LIN {X 0.167,Y -651.336,Z 1359.331,A 0.000,B 0.000,C 90.000,E1 95.511} C_DIS
LIN {X 0.159,Y -645.821,Z 1359.326,A 0.000,B 0.000,C 90.000,E1 94.645} C_DIS
LIN {X 0.149,Y -640.696,Z 1359.322,A 0.000,B 0.000,C 90.000,E1 93.898} C_DIS
LIN {X 0.299,Y -636.929,Z 1359.319,A 0.000,B 0.000,C 90.000,E1 93.383} C_DIS
LIN {X -0.288,Y -631.276,Z 1359.316,A 0.000,B 0.000,C 90.000,E1 92.808} C_DIS
LIN {X -0.177,Y -625.115,Z 1359.312,A 0.000,B 0.000,C 90.000,E1 92.178} C_DIS
LIN {X -0.172,Y -616.219,Z 1359.307,A 0.000,B 0.000,C 90.000,E1 91.318} C_DIS
LIN {X 0.233,Y -610.785,Z 1359.305,A 0.000,B 0.000,C 90.000,E1 90.802} C_DIS
LIN {X 0.209,Y -607.830,Z 1359.303,A 0.000,B 0.000,C 90.000,E1 90.573} C_DIS
LIN {X -0.246,Y -603.158,Z 1359.302,A 0.000,B 0.000,C 90.000,E1 90.286} C_DIS
LIN {X -0.039,Y -596.420,Z 1359.299,A 0.000,B 0.000,C 90.000,E1 89.885} C_DIS
LIN {X -0.028,Y -592.860,Z 1359.298,A 0.000,B 0.000,C 90.000,E1 89.714} C_DIS
LIN {X -0.153,Y -585.830,Z 1359.297,A 0.000,B 0.000,C 90.000,E1 89.427} C_DIS
LIN {X 0.188,Y -582.520,Z 1359.296,A 0.000,B 0.000,C 90.000,E1 89.255} C_DIS
LIN {X -0.070,Y -578.389,Z 1359.295,A 0.000,B 0.000,C 90.000,E1 89.083} C_DIS
LIN {X 0.000,Y -574.152,Z 1359.293,A 0.000,B 0.000,C 90.000,E1 88.797} C_DIS
LIN {X -0.034,Y -574.128,Z 1359.293,A 0.000,B 0.000,C 90.000,E1 88.797} C_DIS
LIN {X 0.004,Y -573.399,Z 1359.292,A 0.000,B 0.000,C 90.000,E1 88.625} C_DIS
LIN {X -0.160,Y -573.188,Z 1359.290,A 0.000,B 0.000,C 90.000,E1 88.165} C_DIS
LIN {X 0.226,Y -575.527,Z 1359.275,A 0.000,B 0.000,C 90.000,E1 85.412} C_DIS
LIN {X 0.222,Y -577.636,Z 1359.264,A 0.000,B 0.000,C 90.000,E1 83.514} C_DIS
LIN {X -0.164,Y -579.848,Z 1359.254,A 0.000,B 0.000,C 90.000,E1 81.659} C_DIS
LIN {X 0.201,Y -581.498,Z 1359.246,A 0.000,B 0.000,C 90.000,E1 80.274} C_DIS
LIN {X 0.218,Y -582.949,Z 1359.239,A 0.000,B 0.000,C 90.000,E1 78.926} C_DIS
LIN {X -0.092,Y -584.010,Z 1359.233,A 0.000,B 0.000,C 90.000,E1 77.881} C_DIS
LIN {X -0.220,Y -585.490,Z 1359.224,A 0.000,B 0.000,C 90.000,E1 76.284} C_DIS
LIN {X -0.138,Y -586.504,Z 1359.216,A 0.000,B 0.000,C 90.000,E1 74.936} C_DIS
LIN {X -0.144,Y -587.223,Z 1359.210,A 0.000,B 0.000,C 90.000,E1 73.866} C_DIS
LIN {X -0.199,Y -588.435,Z 1359.200,A 0.000,B 0.000,C 90.000,E1 72.000} C_DIS
LIN {X 0.200,Y -589.644,Z 1359.188,A 0.000,B 0.000,C 90.000,E1 69.826} C_DIS
LIN {X -0.062,Y -590.952,Z 1359.176,A 0.000,B 0.000,C 90.000,E1 67.720} C_DIS
LIN {X 0.061,Y -592.317,Z 1359.166,A 0.000,B 0.000,C 90.000,E1 65.845} C_DIS
LIN {X -0.139,Y -593.439,Z 1359.159,A 0.000,B 0.000,C 90.000,E1 64.537} C_DIS
LIN {X 0.099,Y -594.582,Z 1359.150,A 0.000,B 0.000,C 90.000,E1 62.922} C_DIS
LIN {X 0.280,Y -596.052,Z 1359.139,A 0.000,B 0.000,C 90.000,E1 61.051} C_DIS
LIN {X 0.132,Y -597.309,Z 1359.132,A 0.000,B 0.000,C 90.000,E1 59.744} C_DIS
LIN {X -0.208,Y -598.613,Z 1359.125,A 0.000,B 0.000,C 90.000,E1 58.456} C_DIS
LIN {X 0.220,Y -600.158,Z 1359.116,A 0.000,B 0.000,C 90.000,E1 56.834} C_DIS
LIN {X 0.018,Y -601.130,Z 1359.110,A 0.000,B 0.000,C 90.000,E1 55.801} C_DIS
LIN {X 0.327,Y -602.568,Z 1359.101,A 0.000,B 0.000,C 90.000,E1 54.196} C_DIS
LIN {X -0.341,Y -603.576,Z 1359.095,A 0.000,B 0.000,C 90.000,E1 53.210} C_DIS
LIN {X 0.213,Y -604.481,Z 1359.090,A 0.000,B 0.000,C 90.000,E1 52.110} C_DIS
LIN {X 0.196,Y -605.361,Z 1359.082,A 0.000,B 0.000,C 90.000,E1 50.803} C_DIS
LIN {X -0.282,Y -606.128,Z 1359.075,A 0.000,B 0.000,C 90.000,E1 49.542} C_DIS
LIN {X -0.159,Y -606.615,Z 1359.069,A 0.000,B 0.000,C 90.000,E1 48.485} C_DIS
LIN {X -0.007,Y -607.015,Z 1359.061,A 0.000,B 0.000,C 90.000,E1 46.905} C_DIS
LIN {X 0.160,Y -607.095,Z 1359.052,A 0.000,B 0.000,C 90.000,E1 45.324} C_DIS
LIN {X 0.266,Y -607.003,Z 1359.046,A 0.000,B 0.000,C 90.000,E1 44.271} C_DIS
LIN {X -0.051,Y -606.655,Z 1359.040,A 0.000,B 0.000,C 90.000,E1 43.257} C_DIS
LIN {X 0.100,Y -605.947,Z 1359.032,A 0.000,B 0.000,C 90.000,E1 41.676} C_DIS
LIN {X 0.220,Y -605.426,Z 1359.026,A 0.000,B 0.000,C 90.000,E1 40.620} C_DIS
LIN {X 0.004,Y -604.489,Z 1359.017,A 0.000,B 0.000,C 90.000,E1 39.072} C_DIS
LIN {X 0.356,Y -603.496,Z 1359.010,A 0.000,B 0.000,C 90.000,E1 37.729} C_DIS
LIN {X 0.283,Y -602.735,Z 1359.005,A 0.000,B 0.000,C 90.000,E1 36.950} C_DIS
LIN {X 0.206,Y -601.887,Z 1359.001,A 0.000,B 0.000,C 90.000,E1 36.171} C_DIS
LIN {X 0.120,Y -600.627,Z 1358.997,A 0.000,B 0.000,C 90.000,E1 35.391} C_DIS
LIN {X 0.019,Y -599.217,Z 1358.992,A 0.000,B 0.000,C 90.000,E1 34.612} C_DIS
LIN {X -0.200,Y -597.011,Z 1358.986,A 0.000,B 0.000,C 90.000,E1 33.579} C_DIS
LIN {X 0.269,Y -593.830,Z 1358.979,A 0.000,B 0.000,C 90.000,E1 32.212} C_DIS
LIN {X -0.129,Y -592.363,Z 1358.976,A 0.000,B 0.000,C 90.000,E1 31.720} C_DIS
LIN {X -0.253,Y -588.851,Z 1358.970,A 0.000,B 0.000,C 90.000,E1 30.669} C_DIS
LIN {X -0.299,Y -585.983,Z 1358.966,A 0.000,B 0.000,C 90.000,E1 29.873} C_DIS
LIN {X -0.250,Y -583.870,Z 1358.963,A 0.000,B 0.000,C 90.000,E1 29.333} C_DIS
LIN {X 0.157,Y -580.292,Z 1358.958,A 0.000,B 0.000,C 90.000,E1 28.487} C_DIS
LIN {X -0.066,Y -575.633,Z 1358.953,A 0.000,B 0.000,C 90.000,E1 27.564} C_DIS
LIN {X 0.060,Y -572.066,Z 1358.949,A 0.000,B 0.000,C 90.000,E1 26.873} C_DIS
LIN {X -0.266,Y -568.990,Z 1358.946,A 0.000,B 0.000,C 90.000,E1 26.360} C_DIS
LIN {X -0.191,Y -564.804,Z 1358.943,A 0.000,B 0.000,C 90.000,E1 25.668} C_DIS
LIN {X 0.184,Y -561.209,Z 1358.939,A 0.000,B 0.000,C 90.000,E1 25.079} C_DIS
LIN {X -0.103,Y -558.437,Z 1358.937,A 0.000,B 0.000,C 90.000,E1 24.695} C_DIS
LIN {X -0.125,Y -553.412,Z 1358.933,A 0.000,B 0.000,C 90.000,E1 24.003} C_DIS
LIN {X -0.023,Y -546.987,Z 1358.929,A 0.000,B 0.000,C 90.000,E1 23.153} C_DIS
LIN {X -0.015,Y -542.308,Z 1358.926,A 0.000,B 0.000,C 90.000,E1 22.589} C_DIS
LIN {X 0.297,Y -534.020,Z 1358.920,A 0.000,B 0.000,C 90.000,E1 21.589} C_DIS
LIN {X 0.096,Y -523.631,Z 1358.914,A 0.000,B 0.000,C 90.000,E1 20.482} C_DIS
LIN {X -0.092,Y -513.039,Z 1358.908,A 0.000,B 0.000,C 90.000,E1 19.396} C_DIS
LIN {X 0.217,Y -502.297,Z 1358.901,A 0.000,B 0.000,C 90.000,E1 18.236} C_DIS
LIN {X 0.199,Y -493.019,Z 1358.896,A 0.000,B 0.000,C 90.000,E1 17.275} C_DIS
LIN {X 0.067,Y -480.292,Z 1358.889,A 0.000,B 0.000,C 90.000,E1 16.079} C_DIS
LIN {X 0.101,Y -467.549,Z 1358.882,A 0.000,B 0.000,C 90.000,E1 14.828} C_DIS
LIN {X 0.172,Y -457.530,Z 1358.877,A 0.000,B 0.000,C 90.000,E1 13.828} C_DIS
LIN {X 0.113,Y -438.983,Z 1358.867,A 0.000,B 0.000,C 90.000,E1 11.951} C_DIS
LIN {X 0.208,Y -420.924,Z 1358.856,A 0.000,B 0.000,C 90.000,E1 9.962} C_DIS
LIN {X -0.132,Y -406.834,Z 1358.847,A 0.000,B 0.000,C 90.000,E1 8.398} C_DIS
LIN {X 0.062,Y -397.118,Z 1358.840,A 0.000,B 0.000,C 90.000,E1 7.239} C_DIS
LIN {X -0.114,Y -393.534,Z 1358.837,A 0.000,B 0.000,C 90.000,E1 6.720} C_DIS
LIN {X -0.153,Y -393.499,Z 1358.837,A 0.000,B 0.000,C 90.000,E1 6.720} C_DIS
LIN {X 0.105,Y -395.070,Z 1358.836,A 0.000,B 0.000,C 90.000,E1 6.429} C_DIS
LIN {X -0.156,Y -397.982,Z 1358.834,A 0.000,B 0.000,C 90.000,E1 6.201} C_DIS
LIN {X -0.095,Y -401.724,Z 1358.833,A 0.000,B 0.000,C 90.000,E1 5.910} C_DIS
LIN {X -0.107,Y -410.009,Z 1358.830,A 0.000,B 0.000,C 90.000,E1 5.334} C_DIS
LIN {X 0.013,Y -417.658,Z 1358.826,A 0.000,B 0.000,C 90.000,E1 4.702} C_DIS
LIN {X -0.174,Y -423.633,Z 1358.823,A 0.000,B 0.000,C 90.000,E1 4.188} C_DIS
LIN {X -0.069,Y -430.586,Z 1358.819,A 0.000,B 0.000,C 90.000,E1 3.440} C_DIS
LIN {X 0.124,Y -437.371,Z 1358.815,A 0.000,B 0.000,C 90.000,E1 2.636} C_DIS
LIN {X -0.030,Y -442.782,Z 1358.811,A 0.000,B 0.000,C 90.000,E1 2.007} C_DIS
LIN {X -0.066,Y -450.455,Z 1358.806,A 0.000,B 0.000,C 90.000,E1 1.031} C_DIS
LIN {X 0.000,Y -457.754,Z 1358.800,A 0.000,B 0.000,C 90.000,E1 360.000} C_DIS
LIN {X 0.008,Y -462.424,Z 1358.796,A 0.000,B 0.000,C 90.000,E1 359.312} C_DIS
LIN {X 0.077,Y -467.489,Z 1358.792,A 0.000,B 0.000,C 90.000,E1 358.511} C_DIS
LIN {X 0.212,Y -472.140,Z 1358.787,A 0.000,B 0.000,C 90.000,E1 357.707} C_DIS
LIN {X -0.104,Y -476.442,Z 1358.783,A 0.000,B 0.000,C 90.000,E1 356.963} C_DIS
LIN {X -0.018,Y -479.732,Z 1358.780,A 0.000,B 0.000,C 90.000,E1 356.331} C_DIS
LIN {X -0.095,Y -484.122,Z 1358.775,A 0.000,B 0.000,C 90.000,E1 355.412} C_DIS
LIN {X 0.206,Y -487.474,Z 1358.770,A 0.000,B 0.000,C 90.000,E1 354.609} C_DIS
LIN {X 0.226,Y -489.412,Z 1358.768,A 0.000,B 0.000,C 90.000,E1 354.147} C_DIS
LIN {X -0.190,Y -492.808,Z 1358.763,A 0.000,B 0.000,C 90.000,E1 353.280} C_DIS
LIN {X 0.022,Y -494.928,Z 1358.759,A 0.000,B 0.000,C 90.000,E1 352.648} C_DIS
LIN {X -0.176,Y -496.874,Z 1358.756,A 0.000,B 0.000,C 90.000,E1 352.064} C_DIS
LIN {X -0.020,Y -499.436,Z 1358.751,A 0.000,B 0.000,C 90.000,E1 351.141} C_DIS
LIN {X 0.088,Y -502.578,Z 1358.744,A 0.000,B 0.000,C 90.000,E1 349.926} C_DIS
LIN {X -0.109,Y -504.658,Z 1358.739,A 0.000,B 0.000,C 90.000,E1 349.050} C_DIS
LIN {X -0.282,Y -506.462,Z 1358.734,A 0.000,B 0.000,C 90.000,E1 348.173} C_DIS
LIN {X 0.168,Y -508.137,Z 1358.729,A 0.000,B 0.000,C 90.000,E1 347.229} C_DIS
LIN {X 0.069,Y -510.411,Z 1358.721,A 0.000,B 0.000,C 90.000,E1 345.755} C_DIS
LIN {X 0.079,Y -511.492,Z 1358.716,A 0.000,B 0.000,C 90.000,E1 344.866} C_DIS
LIN {X 0.100,Y -512.345,Z 1358.711,A 0.000,B 0.000,C 90.000,E1 343.976} C_DIS
LIN {X 0.126,Y -512.947,Z 1358.706,A 0.000,B 0.000,C 90.000,E1 343.087} C_DIS
LIN {X 0.236,Y -513.014,Z 1358.704,A 0.000,B 0.000,C 90.000,E1 342.779} C_DIS
LIN {X 0.194,Y -512.921,Z 1358.703,A 0.000,B 0.000,C 90.000,E1 342.489} C_DIS
LIN {X -0.182,Y -512.687,Z 1358.701,A 0.000,B 0.000,C 90.000,E1 342.236} C_DIS
LIN {X -0.226,Y -512.193,Z 1358.700,A 0.000,B 0.000,C 90.000,E1 341.945} C_DIS
LIN {X -0.112,Y -511.312,Z 1358.698,A 0.000,B 0.000,C 90.000,E1 341.638} C_DIS
LIN {X 0.186,Y -510.592,Z 1358.697,A 0.000,B 0.000,C 90.000,E1 341.456} C_DIS
LIN {X 0.001,Y -509.317,Z 1358.696,A 0.000,B 0.000,C 90.000,E1 341.329} C_DIS
LIN {X -0.056,Y -501.855,Z 1358.695,A 0.000,B 0.000,C 90.000,E1 341.040} C_DIS
LIN {X 0.071,Y -471.003,Z 1358.688,A 0.000,B 0.000,C 90.000,E1 339.752} C_DIS
LIN {X -0.074,Y -442.137,Z 1358.680,A 0.000,B 0.000,C 90.000,E1 338.411} C_DIS
LIN {X -0.024,Y -416.847,Z 1358.672,A 0.000,B 0.000,C 90.000,E1 337.050} C_DIS
LIN {X 0.105,Y -393.487,Z 1358.665,A 0.000,B 0.000,C 90.000,E1 335.613} C_DIS
LIN {X 0.028,Y -372.048,Z 1358.656,A 0.000,B 0.000,C 90.000,E1 334.152} C_DIS
LIN {X -0.045,Y -364.343,Z 1358.653,A 0.000,B 0.000,C 90.000,E1 333.589} C_DIS
LIN {X -0.070,Y -364.332,Z 1358.653,A 0.000,B 0.000,C 90.000,E1 333.589} C_DIS
LIN {X -0.037,Y -365.965,Z 1358.643,A 0.000,B 0.000,C 90.000,E1 331.691} C_DIS
LIN {X 0.125,Y -366.381,Z 1358.639,A 0.000,B 0.000,C 90.000,E1 330.923} C_DIS
LIN {X 0.067,Y -371.337,Z 1358.604,A 0.000,B 0.000,C 90.000,E1 324.642} C_DIS
LIN {X 0.055,Y -371.755,Z 1358.602,A 0.000,B 0.000,C 90.000,E1 324.276} C_DIS
LIN {X -0.169,Y -377.338,Z 1358.567,A 0.000,B 0.000,C 90.000,E1 318.081} C_DIS
LIN {X 0.111,Y -378.225,Z 1358.563,A 0.000,B 0.000,C 90.000,E1 317.310} C_DIS
LIN {X 0.101,Y -383.920,Z 1358.531,A 0.000,B 0.000,C 90.000,E1 311.515} C_DIS
LIN {X -0.104,Y -384.881,Z 1358.527,A 0.000,B 0.000,C 90.000,E1 310.825} C_DIS
LIN {X -0.183,Y -390.590,Z 1358.495,A 0.000,B 0.000,C 90.000,E1 305.105} C_DIS
LIN {X -0.117,Y -391.084,Z 1358.493,A 0.000,B 0.000,C 90.000,E1 304.739} C_DIS
LIN {X 0.123,Y -391.639,Z 1358.489,A 0.000,B 0.000,C 90.000,E1 303.992} C_DIS
LIN {X 0.019,Y -396.807,Z 1358.459,A 0.000,B 0.000,C 90.000,E1 298.693} C_DIS
LIN {X -0.110,Y -397.114,Z 1358.458,A 0.000,B 0.000,C 90.000,E1 298.359} C_DIS
LIN {X 0.045,Y -401.585,Z 1358.426,A 0.000,B 0.000,C 90.000,E1 292.717} C_DIS
LIN {X -0.064,Y -404.646,Z 1358.395,A 0.000,B 0.000,C 90.000,E1 287.149} C_DIS
LIN {X 0.022,Y -404.736,Z 1358.391,A 0.000,B 0.000,C 90.000,E1 286.441} C_DIS
LIN {X -0.082,Y -406.092,Z 1358.364,A 0.000,B 0.000,C 90.000,E1 281.591} C_DIS
LIN {X -0.075,Y -406.100,Z 1358.362,A 0.000,B 0.000,C 90.000,E1 281.243} C_DIS
LIN {X -0.039,Y -405.676,Z 1358.333,A 0.000,B 0.000,C 90.000,E1 276.030} C_DIS
LIN {X -0.030,Y -405.294,Z 1358.330,A 0.000,B 0.000,C 90.000,E1 275.334} C_DIS
LIN {X 0.040,Y -403.505,Z 1358.305,A 0.000,B 0.000,C 90.000,E1 270.802} C_DIS
LIN {X 0.008,Y -403.297,Z 1358.303,A 0.000,B 0.000,C 90.000,E1 270.458} C_DIS
LIN {X 0.191,Y -398.946,Z 1358.271,A 0.000,B 0.000,C 90.000,E1 264.837} C_DIS
LIN {X 0.059,Y -393.120,Z 1358.242,A 0.000,B 0.000,C 90.000,E1 259.567} C_DIS
LIN {X 0.020,Y -392.850,Z 1358.240,A 0.000,B 0.000,C 90.000,E1 259.218} C_DIS
LIN {X 0.133,Y -386.009,Z 1358.212,A 0.000,B 0.000,C 90.000,E1 254.212} C_DIS
LIN {X 0.074,Y -385.282,Z 1358.208,A 0.000,B 0.000,C 90.000,E1 253.504} C_DIS
LIN {X 0.094,Y -384.794,Z 1358.206,A 0.000,B 0.000,C 90.000,E1 253.142} C_DIS
LIN {X -0.033,Y -377.991,Z 1358.182,A 0.000,B 0.000,C 90.000,E1 248.827} C_DIS
LIN {X 0.054,Y -376.249,Z 1358.174,A 0.000,B 0.000,C 90.000,E1 247.358} C_DIS
LIN {X 0.155,Y -374.973,Z 1358.170,A 0.000,B 0.000,C 90.000,E1 246.613} C_DIS
LIN {X -0.110,Y -368.437,Z 1358.148,A 0.000,B 0.000,C 90.000,E1 242.615} C_DIS
LIN {X 0.193,Y -366.076,Z 1358.138,A 0.000,B 0.000,C 90.000,E1 240.717} C_DIS
LIN {X 0.100,Y -359.217,Z 1358.115,A 0.000,B 0.000,C 90.000,E1 236.628} C_DIS
LIN {X 0.117,Y -355.870,Z 1358.100,A 0.000,B 0.000,C 90.000,E1 233.989} C_DIS
LIN {X -0.078,Y -348.813,Z 1358.075,A 0.000,B 0.000,C 90.000,E1 229.461} C_DIS
LIN {X -0.002,Y -346.201,Z 1358.062,A 0.000,B 0.000,C 90.000,E1 227.148} C_DIS
LIN {X -0.115,Y -345.709,Z 1358.060,A 0.000,B 0.000,C 90.000,E1 226.782} C_DIS
LIN {X -0.153,Y -339.000,Z 1358.032,A 0.000,B 0.000,C 90.000,E1 221.757} C_DIS
LIN {X -0.073,Y -336.856,Z 1358.019,A 0.000,B 0.000,C 90.000,E1 219.402} C_DIS
LIN {X -0.167,Y -330.874,Z 1357.988,A 0.000,B 0.000,C 90.000,E1 213.913} C_DIS
LIN {X -0.038,Y -329.305,Z 1357.975,A 0.000,B 0.000,C 90.000,E1 211.514} C_DIS
LIN {X -0.079,Y -327.813,Z 1357.967,A 0.000,B 0.000,C 90.000,E1 210.001} C_DIS
LIN {X -0.096,Y -327.817,Z 1357.967,A 0.000,B 0.000,C 90.000,E1 210.001} C_DIS
LIN {X -0.055,Y -346.466,Z 1357.957,A 0.000,B 0.000,C 90.000,E1 208.281} C_DIS
LIN {X -0.072,Y -366.391,Z 1357.948,A 0.000,B 0.000,C 90.000,E1 206.668} C_DIS
LIN {X 0.068,Y -388.272,Z 1357.939,A 0.000,B 0.000,C 90.000,E1 205.079} C_DIS
LIN {X -0.030,Y -412.110,Z 1357.931,A 0.000,B 0.000,C 90.000,E1 203.590} C_DIS
LIN {X 0.014,Y -437.913,Z 1357.923,A 0.000,B 0.000,C 90.000,E1 202.153} C_DIS
LIN {X -0.025,Y -446.576,Z 1357.921,A 0.000,B 0.000,C 90.000,E1 201.716} C_DIS
LIN {X 0.048,Y -448.741,Z 1357.920,A 0.000,B 0.000,C 90.000,E1 201.535} C_DIS
LIN {X 0.098,Y -450.176,Z 1357.918,A 0.000,B 0.000,C 90.000,E1 201.280} C_DIS
LIN {X -0.026,Y -451.373,Z 1357.917,A 0.000,B 0.000,C 90.000,E1 200.972} C_DIS
LIN {X -0.143,Y -452.250,Z 1357.915,A 0.000,B 0.000,C 90.000,E1 200.663} C_DIS
LIN {X 0.166,Y -452.894,Z 1357.913,A 0.000,B 0.000,C 90.000,E1 200.301} C_DIS
LIN {X -0.056,Y -453.754,Z 1357.909,A 0.000,B 0.000,C 90.000,E1 199.685} C_DIS
LIN {X -0.127,Y -455.519,Z 1357.899,A 0.000,B 0.000,C 90.000,E1 197.764} C_DIS
LIN {X -0.142,Y -456.369,Z 1357.893,A 0.000,B 0.000,C 90.000,E1 196.804} C_DIS
LIN {X -0.150,Y -457.179,Z 1357.888,A 0.000,B 0.000,C 90.000,E1 195.843} C_DIS
LIN {X 0.171,Y -458.653,Z 1357.877,A 0.000,B 0.000,C 90.000,E1 193.883} C_DIS
LIN {X -0.137,Y -460.081,Z 1357.867,A 0.000,B 0.000,C 90.000,E1 192.007} C_DIS
LIN {X 0.246,Y -461.258,Z 1357.858,A 0.000,B 0.000,C 90.000,E1 190.366} C_DIS
LIN {X 0.032,Y -462.299,Z 1357.849,A 0.000,B 0.000,C 90.000,E1 188.803} C_DIS
LIN {X 0.050,Y -462.908,Z 1357.842,A 0.000,B 0.000,C 90.000,E1 187.530} C_DIS
LIN {X -0.174,Y -463.277,Z 1357.837,A 0.000,B 0.000,C 90.000,E1 186.606} C_DIS
LIN {X 0.055,Y -463.743,Z 1357.828,A 0.000,B 0.000,C 90.000,E1 184.992} C_DIS
LIN {X -0.171,Y -463.876,Z 1357.823,A 0.000,B 0.000,C 90.000,E1 184.069} C_DIS
LIN {X -0.221,Y -463.811,Z 1357.816,A 0.000,B 0.000,C 90.000,E1 182.808} C_DIS
LIN {X -0.057,Y -463.396,Z 1357.807,A 0.000,B 0.000,C 90.000,E1 181.203} C_DIS
LIN {X 0.125,Y -462.817,Z 1357.801,A 0.000,B 0.000,C 90.000,E1 180.229} C_DIS
LIN {X 0.089,Y -462.219,Z 1357.798,A 0.000,B 0.000,C 90.000,E1 179.599} C_DIS
LIN {X -0.204,Y -460.933,Z 1357.793,A 0.000,B 0.000,C 90.000,E1 178.682} C_DIS
LIN {X -0.040,Y -459.392,Z 1357.787,A 0.000,B 0.000,C 90.000,E1 177.707} C_DIS
LIN {X -0.105,Y -458.163,Z 1357.784,A 0.000,B 0.000,C 90.000,E1 177.078} C_DIS
LIN {X -0.156,Y -456.758,Z 1357.780,A 0.000,B 0.000,C 90.000,E1 176.445} C_DIS
LIN {X -0.214,Y -455.001,Z 1357.777,A 0.000,B 0.000,C 90.000,E1 175.812} C_DIS
LIN {X -0.117,Y -451.944,Z 1357.771,A 0.000,B 0.000,C 90.000,E1 174.837} C_DIS
LIN {X -0.210,Y -449.445,Z 1357.768,A 0.000,B 0.000,C 90.000,E1 174.204} C_DIS
LIN {X -0.146,Y -445.112,Z 1357.762,A 0.000,B 0.000,C 90.000,E1 173.223} C_DIS
LIN {X -0.135,Y -439.867,Z 1357.757,A 0.000,B 0.000,C 90.000,E1 172.243} C_DIS
LIN {X -0.126,Y -433.576,Z 1357.751,A 0.000,B 0.000,C 90.000,E1 171.254} C_DIS
LIN {X 0.163,Y -426.639,Z 1357.746,A 0.000,B 0.000,C 90.000,E1 170.218} C_DIS
LIN {X -0.186,Y -415.100,Z 1357.736,A 0.000,B 0.000,C 90.000,E1 168.578} C_DIS
LIN {X 0.103,Y -401.003,Z 1357.724,A 0.000,B 0.000,C 90.000,E1 166.297} C_DIS
LIN {X 0.186,Y -399.048,Z 1357.722,A 0.000,B 0.000,C 90.000,E1 165.936} C_DIS
LIN {X -0.132,Y -396.347,Z 1357.719,A 0.000,B 0.000,C 90.000,E1 165.338} C_DIS
LIN {X 0.045,Y -395.353,Z 1357.717,A 0.000,B 0.000,C 90.000,E1 164.991} C_DIS
LIN {X -0.093,Y -395.343,Z 1357.716,A 0.000,B 0.000,C 90.000,E1 164.810} C_DIS
LIN {X 0.018,Y -395.876,Z 1357.715,A 0.000,B 0.000,C 90.000,E1 164.629} C_DIS
LIN {X -0.073,Y -396.619,Z 1357.713,A 0.000,B 0.000,C 90.000,E1 164.267} C_DIS
LIN {X -0.111,Y -396.650,Z 1357.713,A 0.000,B 0.000,C 90.000,E1 164.267} C_DIS
LIN {X 0.036,Y -398.882,Z 1357.711,A 0.000,B 0.000,C 90.000,E1 163.921} C_DIS
LIN {X -0.104,Y -404.818,Z 1357.707,A 0.000,B 0.000,C 90.000,E1 163.268} C_DIS
LIN {X 0.170,Y -413.283,Z 1357.703,A 0.000,B 0.000,C 90.000,E1 162.417} C_DIS
LIN {X 0.161,Y -430.781,Z 1357.694,A 0.000,B 0.000,C 90.000,E1 160.967} C_DIS
LIN {X 0.139,Y -449.702,Z 1357.686,A 0.000,B 0.000,C 90.000,E1 159.518} C_DIS
LIN {X -0.005,Y -459.030,Z 1357.682,A 0.000,B 0.000,C 90.000,E1 158.827} C_DIS
LIN {X -0.093,Y -466.690,Z 1357.679,A 0.000,B 0.000,C 90.000,E1 158.230} C_DIS
LIN {X 0.102,Y -472.556,Z 1357.676,A 0.000,B 0.000,C 90.000,E1 157.720} C_DIS
LIN {X -0.129,Y -481.487,Z 1357.672,A 0.000,B 0.000,C 90.000,E1 156.975} C_DIS
LIN {X 0.013,Y -488.616,Z 1357.668,A 0.000,B 0.000,C 90.000,E1 156.305} C_DIS
LIN {X -0.202,Y -494.236,Z 1357.665,A 0.000,B 0.000,C 90.000,E1 155.793} C_DIS
LIN {X -0.234,Y -502.426,Z 1357.661,A 0.000,B 0.000,C 90.000,E1 154.973} C_DIS
LIN {X -0.232,Y -507.638,Z 1357.658,A 0.000,B 0.000,C 90.000,E1 154.409} C_DIS
LIN {X 0.092,Y -514.031,Z 1357.654,A 0.000,B 0.000,C 90.000,E1 153.640} C_DIS
LIN {X 0.031,Y -517.720,Z 1357.651,A 0.000,B 0.000,C 90.000,E1 153.204} C_DIS
LIN {X -0.107,Y -523.218,Z 1357.647,A 0.000,B 0.000,C 90.000,E1 152.487} C_DIS
LIN {X -0.036,Y -527.181,Z 1357.644,A 0.000,B 0.000,C 90.000,E1 151.897} C_DIS
LIN {X 0.220,Y -529.914,Z 1357.641,A 0.000,B 0.000,C 90.000,E1 151.435} C_DIS
LIN {X 0.198,Y -533.665,Z 1357.637,A 0.000,B 0.000,C 90.000,E1 150.717} C_DIS
LIN {X 0.351,Y -536.318,Z 1357.634,A 0.000,B 0.000,C 90.000,E1 150.127} C_DIS
LIN {X 0.057,Y -538.546,Z 1357.631,A 0.000,B 0.000,C 90.000,E1 149.587} C_DIS
LIN {X -0.035,Y -541.506,Z 1357.626,A 0.000,B 0.000,C 90.000,E1 148.742} C_DIS
LIN {X -0.296,Y -543.205,Z 1357.623,A 0.000,B 0.000,C 90.000,E1 148.201} C_DIS
LIN {X -0.062,Y -545.317,Z 1357.619,A 0.000,B 0.000,C 90.000,E1 147.327} C_DIS
LIN {X 0.001,Y -546.519,Z 1357.615,A 0.000,B 0.000,C 90.000,E1 146.755} C_DIS
LIN {X 0.272,Y -548.094,Z 1357.611,A 0.000,B 0.000,C 90.000,E1 145.881} C_DIS
LIN {X 0.052,Y -549.013,Z 1357.608,A 0.000,B 0.000,C 90.000,E1 145.341} C_DIS
LIN {X 0.258,Y -550.423,Z 1357.601,A 0.000,B 0.000,C 90.000,E1 144.196} C_DIS
LIN {X -0.280,Y -551.611,Z 1357.595,A 0.000,B 0.000,C 90.000,E1 143.130} C_DIS
LIN {X 0.031,Y -552.687,Z 1357.587,A 0.000,B 0.000,C 90.000,E1 141.698} C_DIS
LIN {X 0.273,Y -553.632,Z 1357.579,A 0.000,B 0.000,C 90.000,E1 140.275} C_DIS
LIN {X 0.248,Y -554.825,Z 1357.569,A 0.000,B 0.000,C 90.000,E1 138.324} C_DIS
LIN {X 0.141,Y -555.694,Z 1357.559,A 0.000,B 0.000,C 90.000,E1 136.662} C_DIS
LIN {X -0.285,Y -556.503,Z 1357.549,A 0.000,B 0.000,C 90.000,E1 134.757} C_DIS
LIN {X 0.096,Y -557.915,Z 1357.538,A 0.000,B 0.000,C 90.000,E1 132.771} C_DIS
LIN {X 0.204,Y -558.964,Z 1357.535,A 0.000,B 0.000,C 90.000,E1 132.204} C_DIS
LIN {X 0.161,Y -558.996,Z 1357.535,A 0.000,B 0.000,C 90.000,E1 132.204} C_DIS
LIN {X 0.054,Y -559.934,Z 1357.534,A 0.000,B 0.000,C 90.000,E1 132.081} C_DIS
LIN {X 0.027,Y -560.824,Z 1357.533,A 0.000,B 0.000,C 90.000,E1 131.919} C_DIS
LIN {X -0.016,Y -560.889,Z 1357.533,A 0.000,B 0.000,C 90.000,E1 131.919} C_DIS
LIN {X -0.284,Y -563.030,Z 1357.532,A 0.000,B 0.000,C 90.000,E1 131.838} C_DIS
LIN {X -0.044,Y -574.484,Z 1357.530,A 0.000,B 0.000,C 90.000,E1 131.472} C_DIS
LIN {X 0.051,Y -577.884,Z 1357.530,A 0.000,B 0.000,C 90.000,E1 131.353} C_DIS
LIN {X 0.162,Y -580.585,Z 1357.529,A 0.000,B 0.000,C 90.000,E1 131.229} C_DIS
LIN {X 0.364,Y -583.531,Z 1357.528,A 0.000,B 0.000,C 90.000,E1 131.067} C_DIS
LIN {X -0.188,Y -589.432,Z 1357.526,A 0.000,B 0.000,C 90.000,E1 130.782} C_DIS
LIN {X -0.214,Y -598.051,Z 1357.523,A 0.000,B 0.000,C 90.000,E1 130.172} C_DIS
LIN {X 0.104,Y -600.758,Z 1357.522,A 0.000,B 0.000,C 90.000,E1 129.930} C_DIS
LIN {X 0.329,Y -604.853,Z 1357.520,A 0.000,B 0.000,C 90.000,E1 129.564} C_DIS
LIN {X -0.004,Y -612.552,Z 1357.516,A 0.000,B 0.000,C 90.000,E1 128.874} C_DIS
LIN {X -0.024,Y -617.550,Z 1357.513,A 0.000,B 0.000,C 90.000,E1 128.382} C_DIS
LIN {X -0.399,Y -625.850,Z 1357.508,A 0.000,B 0.000,C 90.000,E1 127.523} C_DIS
LIN {X -0.128,Y -631.317,Z 1357.505,A 0.000,B 0.000,C 90.000,E1 126.870} C_DIS
LIN {X 0.102,Y -638.548,Z 1357.500,A 0.000,B 0.000,C 90.000,E1 125.964} C_DIS
LIN {X -0.117,Y -644.379,Z 1357.496,A 0.000,B 0.000,C 90.000,E1 125.231} C_DIS
LIN {X -0.128,Y -649.777,Z 1357.492,A 0.000,B 0.000,C 90.000,E1 124.485} C_DIS
LIN {X -0.120,Y -653.882,Z 1357.488,A 0.000,B 0.000,C 90.000,E1 123.865} C_DIS
LIN {X -0.173,Y -656.293,Z 1357.486,A 0.000,B 0.000,C 90.000,E1 123.499} C_DIS
LIN {X 0.000,Y -659.749,Z 1357.483,A 0.000,B 0.000,C 90.000,E1 122.880} C_DIS
LIN {X 0.082,Y -662.899,Z 1357.479,A 0.000,B 0.000,C 90.000,E1 122.260} C_DIS
LIN {X -0.096,Y -666.123,Z 1357.475,A 0.000,B 0.000,C 90.000,E1 121.544} C_DIS
LIN {X -0.039,Y -668.150,Z 1357.473,A 0.000,B 0.000,C 90.000,E1 121.052} C_DIS
LIN {X -0.162,Y -670.581,Z 1357.469,A 0.000,B 0.000,C 90.000,E1 120.335} C_DIS
LIN {X 0.078,Y -672.585,Z 1357.464,A 0.000,B 0.000,C 90.000,E1 119.589} C_DIS
LIN {X -0.171,Y -673.743,Z 1357.462,A 0.000,B 0.000,C 90.000,E1 119.127} C_DIS
LIN {X 0.178,Y -674.513,Z 1357.459,A 0.000,B 0.000,C 90.000,E1 118.615} C_DIS
LIN {X -0.058,Y -674.975,Z 1357.456,A 0.000,B 0.000,C 90.000,E1 118.153} C_DIS
LIN {X -0.112,Y -675.219,Z 1357.452,A 0.000,B 0.000,C 90.000,E1 117.436} C_DIS
LIN {X 0.132,Y -675.112,Z 1357.448,A 0.000,B 0.000,C 90.000,E1 116.693} C_DIS
LIN {X 0.079,Y -674.800,Z 1357.444,A 0.000,B 0.000,C 90.000,E1 115.976} C_DIS
LIN {X -0.273,Y -674.207,Z 1357.440,A 0.000,B 0.000,C 90.000,E1 115.283} C_DIS
LIN {X 0.263,Y -673.129,Z 1357.436,A 0.000,B 0.000,C 90.000,E1 114.515} C_DIS
LIN {X -0.277,Y -671.596,Z 1357.434,A 0.000,B 0.000,C 90.000,E1 114.079} C_DIS
LIN {X -0.107,Y -670.422,Z 1357.432,A 0.000,B 0.000,C 90.000,E1 113.823} C_DIS
LIN {X 0.088,Y -667.134,Z 1357.430,A 0.000,B 0.000,C 90.000,E1 113.334} C_DIS
LIN {X 0.167,Y -665.898,Z 1357.429,A 0.000,B 0.000,C 90.000,E1 113.206} C_DIS
LIN {X 0.311,Y -660.002,Z 1357.427,A 0.000,B 0.000,C 90.000,E1 112.770} C_DIS
LIN {X -0.020,Y -658.012,Z 1357.426,A 0.000,B 0.000,C 90.000,E1 112.695} C_DIS
LIN {X 0.247,Y -655.754,Z 1357.426,A 0.000,B 0.000,C 90.000,E1 112.589} C_DIS
LIN {X -0.277,Y -646.048,Z 1357.424,A 0.000,B 0.000,C 90.000,E1 112.333} C_DIS
LIN {X -0.056,Y -633.530,Z 1357.422,A 0.000,B 0.000,C 90.000,E1 112.025} C_DIS
LIN {X -0.114,Y -633.556,Z 1357.422,A 0.000,B 0.000,C 90.000,E1 112.025} C_DIS
LIN {X -0.074,Y -635.850,Z 1357.421,A 0.000,B 0.000,C 90.000,E1 111.716} C_DIS
LIN {X -0.211,Y -644.338,Z 1357.415,A 0.000,B 0.000,C 90.000,E1 110.737} C_DIS
LIN {X -0.282,Y -648.936,Z 1357.412,A 0.000,B 0.000,C 90.000,E1 110.120} C_DIS
LIN {X 0.294,Y -652.648,Z 1357.408,A 0.000,B 0.000,C 90.000,E1 109.450} C_DIS
LIN {X 0.116,Y -656.419,Z 1357.404,A 0.000,B 0.000,C 90.000,E1 108.725} C_DIS
LIN {X 0.085,Y -658.693,Z 1357.401,A 0.000,B 0.000,C 90.000,E1 108.236} C_DIS
LIN {X -0.148,Y -662.766,Z 1357.396,A 0.000,B 0.000,C 90.000,E1 107.275} C_DIS
LIN {X -0.341,Y -664.701,Z 1357.393,A 0.000,B 0.000,C 90.000,E1 106.804} C_DIS
LIN {X 0.226,Y -667.217,Z 1357.389,A 0.000,B 0.000,C 90.000,E1 106.024} C_DIS
LIN {X 0.069,Y -668.744,Z 1357.386,A 0.000,B 0.000,C 90.000,E1 105.552} C_DIS
LIN {X 0.026,Y -670.480,Z 1357.382,A 0.000,B 0.000,C 90.000,E1 104.828} C_DIS
LIN {X -0.112,Y -671.443,Z 1357.380,A 0.000,B 0.000,C 90.000,E1 104.356} C_DIS
LIN {X -0.241,Y -672.173,Z 1357.377,A 0.000,B 0.000,C 90.000,E1 103.883} C_DIS
LIN {X 0.226,Y -672.845,Z 1357.373,A 0.000,B 0.000,C 90.000,E1 103.119} C_DIS
LIN {X 0.044,Y -673.073,Z 1357.369,A 0.000,B 0.000,C 90.000,E1 102.411} C_DIS
LIN {X -0.218,Y -673.039,Z 1357.366,A 0.000,B 0.000,C 90.000,E1 101.951} C_DIS
LIN {X 0.259,Y -672.514,Z 1357.362,A 0.000,B 0.000,C 90.000,E1 101.186} C_DIS
LIN {X 0.129,Y -671.979,Z 1357.360,A 0.000,B 0.000,C 90.000,E1 100.715} C_DIS
LIN {X -0.060,Y -671.671,Z 1357.358,A 0.000,B 0.000,C 90.000,E1 100.489} C_DIS
LIN {X -0.197,Y -670.759,Z 1357.356,A 0.000,B 0.000,C 90.000,E1 100.018} C_DIS
LIN {X 0.206,Y -669.583,Z 1357.353,A 0.000,B 0.000,C 90.000,E1 99.500} C_DIS
LIN {X 0.049,Y -668.134,Z 1357.350,A 0.000,B 0.000,C 90.000,E1 99.029} C_DIS
LIN {X -0.223,Y -666.452,Z 1357.348,A 0.000,B 0.000,C 90.000,E1 98.568} C_DIS
LIN {X 0.059,Y -663.626,Z 1357.344,A 0.000,B 0.000,C 90.000,E1 97.814} C_DIS
LIN {X 0.225,Y -660.258,Z 1357.339,A 0.000,B 0.000,C 90.000,E1 97.068} C_DIS
LIN {X -0.315,Y -655.972,Z 1357.335,A 0.000,B 0.000,C 90.000,E1 96.258} C_DIS
LIN {X -0.218,Y -651.744,Z 1357.331,A 0.000,B 0.000,C 90.000,E1 95.511} C_DIS
LIN {X -0.218,Y -646.238,Z 1357.326,A 0.000,B 0.000,C 90.000,E1 94.645} C_DIS
LIN {X -0.221,Y -641.068,Z 1357.322,A 0.000,B 0.000,C 90.000,E1 93.898} C_DIS
LIN {X -0.066,Y -637.275,Z 1357.319,A 0.000,B 0.000,C 90.000,E1 93.383} C_DIS
LIN {X 0.100,Y -632.801,Z 1357.316,A 0.000,B 0.000,C 90.000,E1 92.865} C_DIS
LIN {X 0.066,Y -625.374,Z 1357.312,A 0.000,B 0.000,C 90.000,E1 92.121} C_DIS
LIN {X 0.086,Y -616.519,Z 1357.307,A 0.000,B 0.000,C 90.000,E1 91.260} C_DIS
LIN {X -0.164,Y -609.678,Z 1357.304,A 0.000,B 0.000,C 90.000,E1 90.688} C_DIS
LIN {X 0.024,Y -603.418,Z 1357.301,A 0.000,B 0.000,C 90.000,E1 90.229} C_DIS
LIN {X 0.275,Y -599.881,Z 1357.300,A 0.000,B 0.000,C 90.000,E1 90.000} C_DIS
LIN {X -0.041,Y -595.108,Z 1357.299,A 0.000,B 0.000,C 90.000,E1 89.771} C_DIS
LIN {X 0.208,Y -586.322,Z 1357.297,A 0.000,B 0.000,C 90.000,E1 89.370} C_DIS
LIN {X -0.035,Y -582.959,Z 1357.296,A 0.000,B 0.000,C 90.000,E1 89.255} C_DIS
LIN {X 0.174,Y -578.518,Z 1357.295,A 0.000,B 0.000,C 90.000,E1 89.026} C_DIS
LIN {X -0.284,Y -575.857,Z 1357.294,A 0.000,B 0.000,C 90.000,E1 88.912} C_DIS
LIN {X -0.149,Y -574.339,Z 1357.293,A 0.000,B 0.000,C 90.000,E1 88.797} C_DIS
LIN {X -0.179,Y -574.299,Z 1357.293,A 0.000,B 0.000,C 90.000,E1 88.797} C_DIS
LIN {X -0.163,Y -573.318,Z 1357.292,A 0.000,B 0.000,C 90.000,E1 88.625} C_DIS
LIN {X -0.205,Y -573.314,Z 1357.292,A 0.000,B 0.000,C 90.000,E1 88.625} C_DIS
LIN {X -0.086,Y -573.058,Z 1357.290,A 0.000,B 0.000,C 90.000,E1 88.282} C_DIS
LIN {X 0.178,Y -573.628,Z 1357.286,A 0.000,B 0.000,C 90.000,E1 87.364} C_DIS
LIN {X 0.083,Y -575.390,Z 1357.275,A 0.000,B 0.000,C 90.000,E1 85.469} C_DIS
LIN {X 0.281,Y -577.817,Z 1357.263,A 0.000,B 0.000,C 90.000,E1 83.280} C_DIS
LIN {X -0.176,Y -580.042,Z 1357.252,A 0.000,B 0.000,C 90.000,E1 81.432} C_DIS
LIN {X 0.282,Y -581.675,Z 1357.245,A 0.000,B 0.000,C 90.000,E1 80.038} C_DIS
LIN {X -0.041,Y -582.835,Z 1357.239,A 0.000,B 0.000,C 90.000,E1 78.993} C_DIS
LIN {X -0.239,Y -583.896,Z 1357.233,A 0.000,B 0.000,C 90.000,E1 77.937} C_DIS
LIN {X -0.178,Y -585.080,Z 1357.225,A 0.000,B 0.000,C 90.000,E1 76.589} C_DIS
LIN {X -0.203,Y -586.006,Z 1357.219,A 0.000,B 0.000,C 90.000,E1 75.519} C_DIS
LIN {X 0.034,Y -586.952,Z 1357.212,A 0.000,B 0.000,C 90.000,E1 74.157} C_DIS
LIN {X -0.197,Y -588.162,Z 1357.202,A 0.000,B 0.000,C 90.000,E1 72.308} C_DIS
LIN {X -0.140,Y -588.891,Z 1357.194,A 0.000,B 0.000,C 90.000,E1 70.967} C_DIS
LIN {X 0.164,Y -589.846,Z 1357.185,A 0.000,B 0.000,C 90.000,E1 69.337} C_DIS
LIN {X 0.018,Y -591.040,Z 1357.175,A 0.000,B 0.000,C 90.000,E1 67.486} C_DIS
LIN {X 0.132,Y -592.445,Z 1357.165,A 0.000,B 0.000,C 90.000,E1 65.613} C_DIS
LIN {X 0.275,Y -593.313,Z 1357.159,A 0.000,B 0.000,C 90.000,E1 64.537} C_DIS
LIN {X -0.289,Y -594.447,Z 1357.150,A 0.000,B 0.000,C 90.000,E1 62.999} C_DIS
LIN {X 0.079,Y -596.159,Z 1357.138,A 0.000,B 0.000,C 90.000,E1 60.845} C_DIS
LIN {X -0.065,Y -597.408,Z 1357.131,A 0.000,B 0.000,C 90.000,E1 59.537} C_DIS
LIN {X 0.197,Y -598.500,Z 1357.125,A 0.000,B 0.000,C 90.000,E1 58.456} C_DIS
LIN {X 0.032,Y -600.287,Z 1357.115,A 0.000,B 0.000,C 90.000,E1 56.628} C_DIS
LIN {X -0.168,Y -601.231,Z 1357.109,A 0.000,B 0.000,C 90.000,E1 55.595} C_DIS
LIN {X -0.011,Y -602.242,Z 1357.103,A 0.000,B 0.000,C 90.000,E1 54.529} C_DIS
LIN {X 0.061,Y -603.464,Z 1357.096,A 0.000,B 0.000,C 90.000,E1 53.210} C_DIS
LIN {X -0.234,Y -604.398,Z 1357.090,A 0.000,B 0.000,C 90.000,E1 52.190} C_DIS
LIN {X 0.335,Y -605.117,Z 1357.084,A 0.000,B 0.000,C 90.000,E1 51.090} C_DIS
LIN {X 0.061,Y -605.759,Z 1357.078,A 0.000,B 0.000,C 90.000,E1 50.070} C_DIS
LIN {X 0.180,Y -606.324,Z 1357.072,A 0.000,B 0.000,C 90.000,E1 49.013} C_DIS
LIN {X 0.046,Y -606.623,Z 1357.068,A 0.000,B 0.000,C 90.000,E1 48.243} C_DIS
LIN {X -0.022,Y -606.960,Z 1357.061,A 0.000,B 0.000,C 90.000,E1 46.944} C_DIS
LIN {X -0.301,Y -607.035,Z 1357.052,A 0.000,B 0.000,C 90.000,E1 45.405} C_DIS
LIN {X -0.196,Y -606.968,Z 1357.046,A 0.000,B 0.000,C 90.000,E1 44.352} C_DIS
LIN {X -0.096,Y -606.629,Z 1357.041,A 0.000,B 0.000,C 90.000,E1 43.299} C_DIS
LIN {X -0.102,Y -605.812,Z 1357.030,A 0.000,B 0.000,C 90.000,E1 41.472} C_DIS
LIN {X -0.239,Y -605.413,Z 1357.026,A 0.000,B 0.000,C 90.000,E1 40.701} C_DIS
LIN {X -0.072,Y -604.512,Z 1357.017,A 0.000,B 0.000,C 90.000,E1 39.116} C_DIS
LIN {X 0.162,Y -603.351,Z 1357.009,A 0.000,B 0.000,C 90.000,E1 37.523} C_DIS
LIN {X 0.113,Y -601.947,Z 1357.001,A 0.000,B 0.000,C 90.000,E1 36.217} C_DIS
LIN {X 0.023,Y -600.748,Z 1356.997,A 0.000,B 0.000,C 90.000,E1 35.438} C_DIS
LIN {X -0.180,Y -598.777,Z 1356.991,A 0.000,B 0.000,C 90.000,E1 34.405} C_DIS
LIN {X 0.193,Y -597.140,Z 1356.987,A 0.000,B 0.000,C 90.000,E1 33.579} C_DIS
LIN {X -0.158,Y -593.987,Z 1356.979,A 0.000,B 0.000,C 90.000,E1 32.291} C_DIS
LIN {X -0.047,Y -592.541,Z 1356.976,A 0.000,B 0.000,C 90.000,E1 31.750} C_DIS
LIN {X 0.139,Y -589.028,Z 1356.970,A 0.000,B 0.000,C 90.000,E1 30.669} C_DIS
LIN {X 0.095,Y -586.244,Z 1356.966,A 0.000,B 0.000,C 90.000,E1 29.873} C_DIS
LIN {X 0.143,Y -584.129,Z 1356.963,A 0.000,B 0.000,C 90.000,E1 29.333} C_DIS
LIN {X -0.093,Y -579.286,Z 1356.957,A 0.000,B 0.000,C 90.000,E1 28.281} C_DIS
LIN {X -0.162,Y -573.835,Z 1356.951,A 0.000,B 0.000,C 90.000,E1 27.206} C_DIS
LIN {X 0.210,Y -570.128,Z 1356.947,A 0.000,B 0.000,C 90.000,E1 26.488} C_DIS
LIN {X 0.203,Y -565.167,Z 1356.943,A 0.000,B 0.000,C 90.000,E1 25.668} C_DIS
LIN {X -0.168,Y -561.595,Z 1356.940,A 0.000,B 0.000,C 90.000,E1 25.155} C_DIS
LIN {X -0.053,Y -557.768,Z 1356.937,A 0.000,B 0.000,C 90.000,E1 24.591} C_DIS
LIN {X -0.075,Y -552.729,Z 1356.933,A 0.000,B 0.000,C 90.000,E1 23.898} C_DIS
LIN {X -0.143,Y -547.398,Z 1356.929,A 0.000,B 0.000,C 90.000,E1 23.206} C_DIS
LIN {X -0.133,Y -542.779,Z 1356.926,A 0.000,B 0.000,C 90.000,E1 22.642} C_DIS
LIN {X -0.099,Y -533.190,Z 1356.920,A 0.000,B 0.000,C 90.000,E1 21.535} C_DIS
LIN {X -0.117,Y -524.174,Z 1356.914,A 0.000,B 0.000,C 90.000,E1 20.556} C_DIS
LIN {X 0.222,Y -512.202,Z 1356.907,A 0.000,B 0.000,C 90.000,E1 19.268} C_DIS
LIN {X 0.012,Y -502.880,Z 1356.902,A 0.000,B 0.000,C 90.000,E1 18.308} C_DIS
LIN {X -0.061,Y -493.378,Z 1356.896,A 0.000,B 0.000,C 90.000,E1 17.330} C_DIS
LIN {X -0.151,Y -481.952,Z 1356.890,A 0.000,B 0.000,C 90.000,E1 16.260} C_DIS
LIN {X 0.055,Y -470.548,Z 1356.884,A 0.000,B 0.000,C 90.000,E1 15.134} C_DIS
LIN {X -0.175,Y -460.554,Z 1356.879,A 0.000,B 0.000,C 90.000,E1 14.175} C_DIS
LIN {X 0.247,Y -440.645,Z 1356.868,A 0.000,B 0.000,C 90.000,E1 12.119} C_DIS
LIN {X 0.039,Y -421.075,Z 1356.856,A 0.000,B 0.000,C 90.000,E1 10.018} C_DIS
LIN {X 0.106,Y -406.964,Z 1356.847,A 0.000,B 0.000,C 90.000,E1 8.398} C_DIS
LIN {X 0.172,Y -398.490,Z 1356.841,A 0.000,B 0.000,C 90.000,E1 7.409} C_DIS
LIN {X -0.201,Y -395.921,Z 1356.839,A 0.000,B 0.000,C 90.000,E1 7.125} C_DIS
LIN {X 0.187,Y -393.748,Z 1356.838,A 0.000,B 0.000,C 90.000,E1 6.720} C_DIS
LIN {X 0.149,Y -393.744,Z 1356.838,A 0.000,B 0.000,C 90.000,E1 6.720} C_DIS
LIN {X -0.110,Y -394.986,Z 1356.836,A 0.000,B 0.000,C 90.000,E1 6.543} C_DIS
LIN {X -0.197,Y -398.849,Z 1356.834,A 0.000,B 0.000,C 90.000,E1 6.201} C_DIS
LIN {X -0.133,Y -411.027,Z 1356.830,A 0.000,B 0.000,C 90.000,E1 5.334} C_DIS
LIN {X 0.044,Y -417.162,Z 1356.827,A 0.000,B 0.000,C 90.000,E1 4.821} C_DIS
LIN {X -0.132,Y -423.294,Z 1356.824,A 0.000,B 0.000,C 90.000,E1 4.302} C_DIS
LIN {X -0.008,Y -430.412,Z 1356.820,A 0.000,B 0.000,C 90.000,E1 3.555} C_DIS
LIN {X 0.188,Y -437.284,Z 1356.815,A 0.000,B 0.000,C 90.000,E1 2.751} C_DIS
LIN {X 0.145,Y -442.642,Z 1356.812,A 0.000,B 0.000,C 90.000,E1 2.121} C_DIS
LIN {X 0.070,Y -448.720,Z 1356.808,A 0.000,B 0.000,C 90.000,E1 1.375} C_DIS
LIN {X -0.075,Y -453.605,Z 1356.804,A 0.000,B 0.000,C 90.000,E1 0.745} C_DIS
LIN {X 0.000,Y -458.879,Z 1356.800,A 0.000,B 0.000,C 90.000,E1 360.000} C_DIS
LIN {X 0.014,Y -463.554,Z 1356.796,A 0.000,B 0.000,C 90.000,E1 359.312} C_DIS
LIN {X 0.094,Y -468.621,Z 1356.792,A 0.000,B 0.000,C 90.000,E1 358.511} C_DIS
LIN {X 0.241,Y -473.241,Z 1356.787,A 0.000,B 0.000,C 90.000,E1 357.707} C_DIS
LIN {X -0.065,Y -477.577,Z 1356.783,A 0.000,B 0.000,C 90.000,E1 356.963} C_DIS
LIN {X 0.172,Y -481.604,Z 1356.779,A 0.000,B 0.000,C 90.000,E1 356.159} C_DIS
LIN {X -0.034,Y -485.268,Z 1356.775,A 0.000,B 0.000,C 90.000,E1 355.412} C_DIS
LIN {X -0.207,Y -488.615,Z 1356.770,A 0.000,B 0.000,C 90.000,E1 354.666} C_DIS
LIN {X -0.181,Y -490.550,Z 1356.768,A 0.000,B 0.000,C 90.000,E1 354.204} C_DIS
LIN {X -0.097,Y -493.937,Z 1356.763,A 0.000,B 0.000,C 90.000,E1 353.280} C_DIS
LIN {X 0.027,Y -497.049,Z 1356.758,A 0.000,B 0.000,C 90.000,E1 352.356} C_DIS
LIN {X -0.064,Y -498.073,Z 1356.756,A 0.000,B 0.000,C 90.000,E1 352.064} C_DIS
LIN {X 0.106,Y -500.617,Z 1356.751,A 0.000,B 0.000,C 90.000,E1 351.141} C_DIS
LIN {X -0.263,Y -503.735,Z 1356.744,A 0.000,B 0.000,C 90.000,E1 349.982} C_DIS
LIN {X -0.007,Y -506.438,Z 1356.738,A 0.000,B 0.000,C 90.000,E1 348.757} C_DIS
LIN {X -0.161,Y -508.206,Z 1356.733,A 0.000,B 0.000,C 90.000,E1 347.881} C_DIS
LIN {X -0.185,Y -509.777,Z 1356.728,A 0.000,B 0.000,C 90.000,E1 346.992} C_DIS
LIN {X 0.239,Y -511.958,Z 1356.719,A 0.000,B 0.000,C 90.000,E1 345.463} C_DIS
LIN {X -0.230,Y -513.009,Z 1356.714,A 0.000,B 0.000,C 90.000,E1 344.629} C_DIS
LIN {X -0.194,Y -513.816,Z 1356.710,A 0.000,B 0.000,C 90.000,E1 343.740} C_DIS
LIN {X -0.003,Y -514.268,Z 1356.705,A 0.000,B 0.000,C 90.000,E1 342.834} C_DIS
LIN {X 0.079,Y -514.448,Z 1356.701,A 0.000,B 0.000,C 90.000,E1 342.236} C_DIS
LIN {X 0.040,Y -514.379,Z 1356.700,A 0.000,B 0.000,C 90.000,E1 341.945} C_DIS
LIN {X 0.160,Y -514.183,Z 1356.698,A 0.000,B 0.000,C 90.000,E1 341.638} C_DIS
LIN {X 0.117,Y -513.768,Z 1356.697,A 0.000,B 0.000,C 90.000,E1 341.348} C_DIS
LIN {X -0.249,Y -513.042,Z 1356.695,A 0.000,B 0.000,C 90.000,E1 341.094} C_DIS
LIN {X 0.053,Y -512.519,Z 1356.694,A 0.000,B 0.000,C 90.000,E1 340.913} C_DIS
LIN {X -0.128,Y -511.799,Z 1356.693,A 0.000,B 0.000,C 90.000,E1 340.786} C_DIS
LIN {X 0.171,Y -510.613,Z 1356.692,A 0.000,B 0.000,C 90.000,E1 340.604} C_DIS
LIN {X -0.181,Y -507.406,Z 1356.692,A 0.000,B 0.000,C 90.000,E1 340.496} C_DIS
LIN {X 0.030,Y -476.133,Z 1356.684,A 0.000,B 0.000,C 90.000,E1 339.156} C_DIS
LIN {X -0.144,Y -447.363,Z 1356.677,A 0.000,B 0.000,C 90.000,E1 337.794} C_DIS
LIN {X -0.075,Y -422.178,Z 1356.669,A 0.000,B 0.000,C 90.000,E1 336.410} C_DIS
LIN {X -0.066,Y -398.933,Z 1356.661,A 0.000,B 0.000,C 90.000,E1 334.973} C_DIS
LIN {X 0.099,Y -377.610,Z 1356.653,A 0.000,B 0.000,C 90.000,E1 333.461} C_DIS
LIN {X -0.107,Y -365.194,Z 1356.647,A 0.000,B 0.000,C 90.000,E1 332.538} C_DIS
LIN {X -0.132,Y -365.195,Z 1356.647,A 0.000,B 0.000,C 90.000,E1 332.538} C_DIS
LIN {X 0.085,Y -366.045,Z 1356.642,A 0.000,B 0.000,C 90.000,E1 331.591} C_DIS
LIN {X -0.209,Y -367.179,Z 1356.630,A 0.000,B 0.000,C 90.000,E1 329.410} C_DIS
LIN {X 0.048,Y -371.805,Z 1356.601,A 0.000,B 0.000,C 90.000,E1 324.196} C_DIS
LIN {X -0.165,Y -377.441,Z 1356.567,A 0.000,B 0.000,C 90.000,E1 318.000} C_DIS
LIN {X 0.116,Y -378.275,Z 1356.563,A 0.000,B 0.000,C 90.000,E1 317.229} C_DIS
LIN {X 0.111,Y -384.027,Z 1356.530,A 0.000,B 0.000,C 90.000,E1 311.434} C_DIS
LIN {X 0.198,Y -384.935,Z 1356.526,A 0.000,B 0.000,C 90.000,E1 310.701} C_DIS
LIN {X -0.174,Y -390.697,Z 1356.495,A 0.000,B 0.000,C 90.000,E1 305.025} C_DIS
LIN {X 0.214,Y -391.195,Z 1356.493,A 0.000,B 0.000,C 90.000,E1 304.612} C_DIS
LIN {X 0.021,Y -396.910,Z 1356.459,A 0.000,B 0.000,C 90.000,E1 298.615} C_DIS
LIN {X -0.106,Y -397.908,Z 1356.449,A 0.000,B 0.000,C 90.000,E1 296.873} C_DIS
LIN {X 0.032,Y -401.638,Z 1356.426,A 0.000,B 0.000,C 90.000,E1 292.642} C_DIS
LIN {X 0.168,Y -404.713,Z 1356.395,A 0.000,B 0.000,C 90.000,E1 287.040} C_DIS
LIN {X 0.171,Y -406.136,Z 1356.364,A 0.000,B 0.000,C 90.000,E1 281.478} C_DIS
LIN {X -0.132,Y -405.443,Z 1356.347,A 0.000,B 0.000,C 90.000,E1 278.398} C_DIS
LIN {X -0.135,Y -405.688,Z 1356.333,A 0.000,B 0.000,C 90.000,E1 275.967} C_DIS
LIN {X -0.064,Y -403.574,Z 1356.306,A 0.000,B 0.000,C 90.000,E1 271.088} C_DIS
LIN {X -0.129,Y -403.240,Z 1356.302,A 0.000,B 0.000,C 90.000,E1 270.401} C_DIS
LIN {X 0.109,Y -399.092,Z 1356.273,A 0.000,B 0.000,C 90.000,E1 265.122} C_DIS
LIN {X 0.051,Y -398.856,Z 1356.271,A 0.000,B 0.000,C 90.000,E1 264.780} C_DIS
LIN {X -0.051,Y -393.337,Z 1356.244,A 0.000,B 0.000,C 90.000,E1 259.859} C_DIS
LIN {X -0.129,Y -392.758,Z 1356.240,A 0.000,B 0.000,C 90.000,E1 259.162} C_DIS
LIN {X -0.050,Y -386.309,Z 1356.214,A 0.000,B 0.000,C 90.000,E1 254.519} C_DIS
LIN {X -0.089,Y -385.206,Z 1356.208,A 0.000,B 0.000,C 90.000,E1 253.449} C_DIS
LIN {X -0.048,Y -383.993,Z 1356.204,A 0.000,B 0.000,C 90.000,E1 252.725} C_DIS
LIN {X -0.219,Y -377.433,Z 1356.180,A 0.000,B 0.000,C 90.000,E1 248.411} C_DIS
LIN {X 0.019,Y -376.160,Z 1356.174,A 0.000,B 0.000,C 90.000,E1 247.283} C_DIS
LIN {X -0.136,Y -368.328,Z 1356.147,A 0.000,B 0.000,C 90.000,E1 242.538} C_DIS
LIN {X -0.093,Y -366.466,Z 1356.139,A 0.000,B 0.000,C 90.000,E1 241.051} C_DIS
LIN {X -0.009,Y -365.918,Z 1356.137,A 0.000,B 0.000,C 90.000,E1 240.667} C_DIS
LIN {X 0.080,Y -359.102,Z 1356.114,A 0.000,B 0.000,C 90.000,E1 236.548} C_DIS
LIN {X 0.168,Y -356.246,Z 1356.102,A 0.000,B 0.000,C 90.000,E1 234.276} C_DIS
LIN {X 0.098,Y -355.718,Z 1356.100,A 0.000,B 0.000,C 90.000,E1 233.909} C_DIS
LIN {X -0.099,Y -348.707,Z 1356.074,A 0.000,B 0.000,C 90.000,E1 229.380} C_DIS
LIN {X -0.024,Y -346.116,Z 1356.062,A 0.000,B 0.000,C 90.000,E1 227.067} C_DIS
LIN {X -0.038,Y -342.669,Z 1356.049,A 0.000,B 0.000,C 90.000,E1 224.757} C_DIS
LIN {X 0.156,Y -336.754,Z 1356.018,A 0.000,B 0.000,C 90.000,E1 219.277} C_DIS
LIN {X 0.065,Y -330.807,Z 1355.988,A 0.000,B 0.000,C 90.000,E1 213.785} C_DIS
LIN {X 0.022,Y -329.253,Z 1355.975,A 0.000,B 0.000,C 90.000,E1 211.416} C_DIS
LIN {X 0.128,Y -328.983,Z 1355.973,A 0.000,B 0.000,C 90.000,E1 211.131} C_DIS
LIN {X 0.110,Y -328.994,Z 1355.973,A 0.000,B 0.000,C 90.000,E1 211.131} C_DIS
LIN {X 0.090,Y -346.413,Z 1355.964,A 0.000,B 0.000,C 90.000,E1 209.461} C_DIS
LIN {X 0.169,Y -366.120,Z 1355.954,A 0.000,B 0.000,C 90.000,E1 207.769} C_DIS
LIN {X 0.074,Y -387.777,Z 1355.945,A 0.000,B 0.000,C 90.000,E1 206.155} C_DIS
LIN {X 0.065,Y -411.412,Z 1355.937,A 0.000,B 0.000,C 90.000,E1 204.591} C_DIS
LIN {X 0.221,Y -437.038,Z 1355.928,A 0.000,B 0.000,C 90.000,E1 203.078} C_DIS
LIN {X -0.246,Y -447.347,Z 1355.925,A 0.000,B 0.000,C 90.000,E1 202.589} C_DIS
LIN {X -0.064,Y -449.078,Z 1355.924,A 0.000,B 0.000,C 90.000,E1 202.386} C_DIS
LIN {X 0.025,Y -450.616,Z 1355.923,A 0.000,B 0.000,C 90.000,E1 202.078} C_DIS
LIN {X -0.099,Y -451.732,Z 1355.921,A 0.000,B 0.000,C 90.000,E1 201.770} C_DIS
LIN {X 0.206,Y -452.579,Z 1355.919,A 0.000,B 0.000,C 90.000,E1 201.408} C_DIS
LIN {X 0.093,Y -453.239,Z 1355.917,A 0.000,B 0.000,C 90.000,E1 201.099} C_DIS
LIN {X -0.124,Y -454.164,Z 1355.914,A 0.000,B 0.000,C 90.000,E1 200.482} C_DIS
LIN {X 0.062,Y -455.648,Z 1355.905,A 0.000,B 0.000,C 90.000,E1 198.852} C_DIS
LIN {X -0.153,Y -457.199,Z 1355.896,A 0.000,B 0.000,C 90.000,E1 197.275} C_DIS
LIN {X 0.058,Y -458.332,Z 1355.889,A 0.000,B 0.000,C 90.000,E1 195.969} C_DIS
LIN {X -0.031,Y -459.835,Z 1355.878,A 0.000,B 0.000,C 90.000,E1 194.064} C_DIS
LIN {X 0.240,Y -461.353,Z 1355.868,A 0.000,B 0.000,C 90.000,E1 192.119} C_DIS
LIN {X -0.100,Y -462.853,Z 1355.857,A 0.000,B 0.000,C 90.000,E1 190.254} C_DIS
LIN {X -0.005,Y -463.754,Z 1355.850,A 0.000,B 0.000,C 90.000,E1 188.973} C_DIS
LIN {X 0.031,Y -464.453,Z 1355.843,A 0.000,B 0.000,C 90.000,E1 187.701} C_DIS
LIN {X 0.078,Y -465.043,Z 1355.836,A 0.000,B 0.000,C 90.000,E1 186.429} C_DIS
LIN {X 0.080,Y -465.458,Z 1355.829,A 0.000,B 0.000,C 90.000,E1 185.163} C_DIS
LIN {X 0.088,Y -465.639,Z 1355.822,A 0.000,B 0.000,C 90.000,E1 183.898} C_DIS
LIN {X 0.066,Y -465.565,Z 1355.815,A 0.000,B 0.000,C 90.000,E1 182.636} C_DIS
LIN {X 0.044,Y -465.284,Z 1355.808,A 0.000,B 0.000,C 90.000,E1 181.375} C_DIS
LIN {X -0.216,Y -464.826,Z 1355.802,A 0.000,B 0.000,C 90.000,E1 180.458} C_DIS
LIN {X -0.017,Y -463.957,Z 1355.797,A 0.000,B 0.000,C 90.000,E1 179.484} C_DIS
LIN {X 0.171,Y -462.809,Z 1355.792,A 0.000,B 0.000,C 90.000,E1 178.511} C_DIS
LIN {X 0.149,Y -461.867,Z 1355.788,A 0.000,B 0.000,C 90.000,E1 177.879} C_DIS
LIN {X 0.103,Y -460.768,Z 1355.785,A 0.000,B 0.000,C 90.000,E1 177.249} C_DIS
LIN {X -0.192,Y -458.684,Z 1355.780,A 0.000,B 0.000,C 90.000,E1 176.331} C_DIS
LIN {X 0.220,Y -457.212,Z 1355.776,A 0.000,B 0.000,C 90.000,E1 175.641} C_DIS
LIN {X 0.165,Y -455.338,Z 1355.772,A 0.000,B 0.000,C 90.000,E1 175.008} C_DIS
LIN {X -0.191,Y -451.910,Z 1355.767,A 0.000,B 0.000,C 90.000,E1 174.090} C_DIS
LIN {X -0.098,Y -447.622,Z 1355.762,A 0.000,B 0.000,C 90.000,E1 173.109} C_DIS
LIN {X 0.149,Y -445.217,Z 1355.759,A 0.000,B 0.000,C 90.000,E1 172.591} C_DIS
LIN {X 0.055,Y -441.584,Z 1355.755,A 0.000,B 0.000,C 90.000,E1 171.951} C_DIS
LIN {X -0.171,Y -438.639,Z 1355.753,A 0.000,B 0.000,C 90.000,E1 171.489} C_DIS
LIN {X 0.152,Y -433.161,Z 1355.748,A 0.000,B 0.000,C 90.000,E1 170.622} C_DIS
LIN {X 0.168,Y -425.048,Z 1355.742,A 0.000,B 0.000,C 90.000,E1 169.454} C_DIS
LIN {X 0.203,Y -413.643,Z 1355.732,A 0.000,B 0.000,C 90.000,E1 167.757} C_DIS
LIN {X 0.059,Y -403.886,Z 1355.724,A 0.000,B 0.000,C 90.000,E1 166.228} C_DIS
LIN {X 0.089,Y -399.309,Z 1355.719,A 0.000,B 0.000,C 90.000,E1 165.353} C_DIS
LIN {X -0.019,Y -397.211,Z 1355.715,A 0.000,B 0.000,C 90.000,E1 164.629} C_DIS
LIN {X -0.057,Y -397.214,Z 1355.715,A 0.000,B 0.000,C 90.000,E1 164.629} C_DIS
LIN {X 0.023,Y -397.538,Z 1355.713,A 0.000,B 0.000,C 90.000,E1 164.283} C_DIS
LIN {X -0.016,Y -397.558,Z 1355.713,A 0.000,B 0.000,C 90.000,E1 164.283} C_DIS
LIN {X -0.024,Y -399.061,Z 1355.711,A 0.000,B 0.000,C 90.000,E1 164.031} C_DIS
LIN {X -0.099,Y -399.896,Z 1355.710,A 0.000,B 0.000,C 90.000,E1 163.866} C_DIS
LIN {X 0.213,Y -405.601,Z 1355.707,A 0.000,B 0.000,C 90.000,E1 163.142} C_DIS
LIN {X -0.196,Y -410.311,Z 1355.704,A 0.000,B 0.000,C 90.000,E1 162.725} C_DIS
LIN {X 0.150,Y -420.675,Z 1355.699,A 0.000,B 0.000,C 90.000,E1 161.764} C_DIS
LIN {X 0.121,Y -443.006,Z 1355.689,A 0.000,B 0.000,C 90.000,E1 160.007} C_DIS
LIN {X -0.095,Y -457.291,Z 1355.683,A 0.000,B 0.000,C 90.000,E1 158.954} C_DIS
LIN {X 0.023,Y -466.299,Z 1355.679,A 0.000,B 0.000,C 90.000,E1 158.230} C_DIS
LIN {X 0.181,Y -472.261,Z 1355.676,A 0.000,B 0.000,C 90.000,E1 157.720} C_DIS
LIN {X -0.030,Y -481.212,Z 1355.672,A 0.000,B 0.000,C 90.000,E1 156.975} C_DIS
LIN {X 0.119,Y -488.398,Z 1355.668,A 0.000,B 0.000,C 90.000,E1 156.305} C_DIS
LIN {X -0.140,Y -495.357,Z 1355.665,A 0.000,B 0.000,C 90.000,E1 155.665} C_DIS
LIN {X -0.225,Y -503.598,Z 1355.660,A 0.000,B 0.000,C 90.000,E1 154.845} C_DIS
LIN {X 0.113,Y -511.298,Z 1355.655,A 0.000,B 0.000,C 90.000,E1 153.948} C_DIS
LIN {X -0.093,Y -516.288,Z 1355.652,A 0.000,B 0.000,C 90.000,E1 153.384} C_DIS
LIN {X 0.093,Y -519.772,Z 1355.650,A 0.000,B 0.000,C 90.000,E1 152.922} C_DIS
LIN {X 0.060,Y -523.030,Z 1355.647,A 0.000,B 0.000,C 90.000,E1 152.487} C_DIS
LIN {X 0.131,Y -526.973,Z 1355.644,A 0.000,B 0.000,C 90.000,E1 151.897} C_DIS
LIN {X 0.132,Y -529.689,Z 1355.642,A 0.000,B 0.000,C 90.000,E1 151.463} C_DIS
LIN {X 0.103,Y -533.480,Z 1355.638,A 0.000,B 0.000,C 90.000,E1 150.745} C_DIS
LIN {X -0.216,Y -536.134,Z 1355.634,A 0.000,B 0.000,C 90.000,E1 150.205} C_DIS
LIN {X -0.059,Y -539.337,Z 1355.630,A 0.000,B 0.000,C 90.000,E1 149.331} C_DIS
LIN {X 0.128,Y -541.324,Z 1355.626,A 0.000,B 0.000,C 90.000,E1 148.742} C_DIS
LIN {X -0.117,Y -543.699,Z 1355.622,A 0.000,B 0.000,C 90.000,E1 147.916} C_DIS
LIN {X 0.098,Y -545.103,Z 1355.619,A 0.000,B 0.000,C 90.000,E1 147.327} C_DIS
LIN {X -0.105,Y -546.846,Z 1355.614,A 0.000,B 0.000,C 90.000,E1 146.501} C_DIS
LIN {X -0.025,Y -547.916,Z 1355.611,A 0.000,B 0.000,C 90.000,E1 145.928} C_DIS
LIN {X -0.195,Y -549.190,Z 1355.606,A 0.000,B 0.000,C 90.000,E1 145.102} C_DIS
LIN {X -0.035,Y -550.232,Z 1355.601,A 0.000,B 0.000,C 90.000,E1 144.242} C_DIS
LIN {X -0.128,Y -551.409,Z 1355.595,A 0.000,B 0.000,C 90.000,E1 143.130} C_DIS
LIN {X 0.116,Y -552.271,Z 1355.589,A 0.000,B 0.000,C 90.000,E1 141.984} C_DIS
LIN {X 0.002,Y -553.265,Z 1355.581,A 0.000,B 0.000,C 90.000,E1 140.598} C_DIS
LIN {X -0.041,Y -554.446,Z 1355.570,A 0.000,B 0.000,C 90.000,E1 138.647} C_DIS
LIN {X -0.104,Y -555.542,Z 1355.559,A 0.000,B 0.000,C 90.000,E1 136.701} C_DIS
LIN {X 0.009,Y -556.887,Z 1355.544,A 0.000,B 0.000,C 90.000,E1 133.905} C_DIS
LIN {X -0.066,Y -557.521,Z 1355.540,A 0.000,B 0.000,C 90.000,E1 133.218} C_DIS
LIN {X 0.050,Y -558.193,Z 1355.538,A 0.000,B 0.000,C 90.000,E1 132.813} C_DIS
LIN {X 0.234,Y -559.458,Z 1355.536,A 0.000,B 0.000,C 90.000,E1 132.447} C_DIS
LIN {X 0.262,Y -559.649,Z 1355.536,A 0.000,B 0.000,C 90.000,E1 132.366} C_DIS
LIN {X 0.220,Y -559.667,Z 1355.536,A 0.000,B 0.000,C 90.000,E1 132.366} C_DIS
LIN {X -0.056,Y -561.318,Z 1355.535,A 0.000,B 0.000,C 90.000,E1 132.285} C_DIS
LIN {X -0.019,Y -567.318,Z 1355.534,A 0.000,B 0.000,C 90.000,E1 132.123} C_DIS
LIN {X 0.060,Y -574.107,Z 1355.533,A 0.000,B 0.000,C 90.000,E1 131.919} C_DIS
LIN {X -0.155,Y -577.345,Z 1355.532,A 0.000,B 0.000,C 90.000,E1 131.838} C_DIS
LIN {X 0.359,Y -579.980,Z 1355.532,A 0.000,B 0.000,C 90.000,E1 131.676} C_DIS
LIN {X -0.270,Y -582.854,Z 1355.531,A 0.000,B 0.000,C 90.000,E1 131.595} C_DIS
LIN {X -0.035,Y -588.808,Z 1355.529,A 0.000,B 0.000,C 90.000,E1 131.229} C_DIS
LIN {X -0.315,Y -591.675,Z 1355.528,A 0.000,B 0.000,C 90.000,E1 131.067} C_DIS
LIN {X -0.300,Y -598.734,Z 1355.525,A 0.000,B 0.000,C 90.000,E1 130.539} C_DIS
LIN {X 0.085,Y -602.809,Z 1355.523,A 0.000,B 0.000,C 90.000,E1 130.172} C_DIS
LIN {X -0.159,Y -608.000,Z 1355.521,A 0.000,B 0.000,C 90.000,E1 129.725} C_DIS
LIN {X -0.202,Y -614.320,Z 1355.517,A 0.000,B 0.000,C 90.000,E1 129.116} C_DIS
LIN {X 0.108,Y -619.218,Z 1355.515,A 0.000,B 0.000,C 90.000,E1 128.588} C_DIS
LIN {X -0.271,Y -627.298,Z 1355.510,A 0.000,B 0.000,C 90.000,E1 127.729} C_DIS
LIN {X -0.072,Y -631.662,Z 1355.507,A 0.000,B 0.000,C 90.000,E1 127.202} C_DIS
LIN {X 0.414,Y -638.595,Z 1355.502,A 0.000,B 0.000,C 90.000,E1 126.297} C_DIS
LIN {X -0.180,Y -644.367,Z 1355.498,A 0.000,B 0.000,C 90.000,E1 125.598} C_DIS
LIN {X -0.247,Y -648.082,Z 1355.495,A 0.000,B 0.000,C 90.000,E1 125.105} C_DIS
LIN {X 0.187,Y -654.058,Z 1355.490,A 0.000,B 0.000,C 90.000,E1 124.199} C_DIS
LIN {X -0.269,Y -658.531,Z 1355.486,A 0.000,B 0.000,C 90.000,E1 123.499} C_DIS
LIN {X 0.305,Y -661.290,Z 1355.483,A 0.000,B 0.000,C 90.000,E1 122.959} C_DIS
LIN {X -0.014,Y -663.791,Z 1355.481,A 0.000,B 0.000,C 90.000,E1 122.498} C_DIS
LIN {X 0.173,Y -666.983,Z 1355.477,A 0.000,B 0.000,C 90.000,E1 121.750} C_DIS
LIN {X -0.185,Y -669.803,Z 1355.473,A 0.000,B 0.000,C 90.000,E1 121.052} C_DIS
LIN {X -0.126,Y -672.858,Z 1355.467,A 0.000,B 0.000,C 90.000,E1 120.079} C_DIS
LIN {X 0.137,Y -674.726,Z 1355.463,A 0.000,B 0.000,C 90.000,E1 119.333} C_DIS
LIN {X 0.083,Y -675.862,Z 1355.459,A 0.000,B 0.000,C 90.000,E1 118.615} C_DIS
LIN {X 0.040,Y -676.376,Z 1355.455,A 0.000,B 0.000,C 90.000,E1 117.897} C_DIS
LIN {X -0.001,Y -676.441,Z 1355.451,A 0.000,B 0.000,C 90.000,E1 117.180} C_DIS
LIN {X -0.158,Y -676.197,Z 1355.446,A 0.000,B 0.000,C 90.000,E1 116.232} C_DIS
LIN {X 0.402,Y -675.679,Z 1355.442,A 0.000,B 0.000,C 90.000,E1 115.463} C_DIS
LIN {X -0.128,Y -675.154,Z 1355.439,A 0.000,B 0.000,C 90.000,E1 115.027} C_DIS
LIN {X 0.238,Y -674.398,Z 1355.436,A 0.000,B 0.000,C 90.000,E1 114.515} C_DIS
LIN {X -0.296,Y -672.867,Z 1355.434,A 0.000,B 0.000,C 90.000,E1 114.079} C_DIS
LIN {X -0.121,Y -671.858,Z 1355.432,A 0.000,B 0.000,C 90.000,E1 113.823} C_DIS
LIN {X -0.053,Y -668.402,Z 1355.430,A 0.000,B 0.000,C 90.000,E1 113.334} C_DIS
LIN {X 0.027,Y -667.281,Z 1355.429,A 0.000,B 0.000,C 90.000,E1 113.206} C_DIS
LIN {X 0.234,Y -661.351,Z 1355.427,A 0.000,B 0.000,C 90.000,E1 112.770} C_DIS
LIN {X 0.033,Y -659.857,Z 1355.426,A 0.000,B 0.000,C 90.000,E1 112.695} C_DIS
LIN {X 0.181,Y -657.500,Z 1355.426,A 0.000,B 0.000,C 90.000,E1 112.589} C_DIS
LIN {X -0.074,Y -652.714,Z 1355.425,A 0.000,B 0.000,C 90.000,E1 112.461} C_DIS
LIN {X -0.031,Y -648.662,Z 1355.424,A 0.000,B 0.000,C 90.000,E1 112.333} C_DIS
LIN {X -0.229,Y -634.430,Z 1355.422,A 0.000,B 0.000,C 90.000,E1 112.025} C_DIS
LIN {X -0.281,Y -634.437,Z 1355.422,A 0.000,B 0.000,C 90.000,E1 112.025} C_DIS
LIN {X 0.171,Y -635.354,Z 1355.422,A 0.000,B 0.000,C 90.000,E1 111.844} C_DIS
LIN {X 0.071,Y -644.817,Z 1355.415,A 0.000,B 0.000,C 90.000,E1 110.737} C_DIS
LIN {X 0.189,Y -649.338,Z 1355.412,A 0.000,B 0.000,C 90.000,E1 110.120} C_DIS
LIN {X -0.021,Y -653.747,Z 1355.408,A 0.000,B 0.000,C 90.000,E1 109.396} C_DIS
LIN {X -0.023,Y -656.868,Z 1355.404,A 0.000,B 0.000,C 90.000,E1 108.779} C_DIS
LIN {X -0.168,Y -660.161,Z 1355.400,A 0.000,B 0.000,C 90.000,E1 108.055} C_DIS
LIN {X 0.252,Y -664.162,Z 1355.395,A 0.000,B 0.000,C 90.000,E1 107.040} C_DIS
LIN {X 0.071,Y -665.978,Z 1355.392,A 0.000,B 0.000,C 90.000,E1 106.567} C_DIS
LIN {X 0.011,Y -668.412,Z 1355.388,A 0.000,B 0.000,C 90.000,E1 105.843} C_DIS
LIN {X -0.065,Y -669.147,Z 1355.387,A 0.000,B 0.000,C 90.000,E1 105.607} C_DIS
LIN {X -0.279,Y -670.884,Z 1355.383,A 0.000,B 0.000,C 90.000,E1 104.898} C_DIS
LIN {X -0.243,Y -671.903,Z 1355.380,A 0.000,B 0.000,C 90.000,E1 104.411} C_DIS
LIN {X 0.219,Y -672.921,Z 1355.376,A 0.000,B 0.000,C 90.000,E1 103.647} C_DIS
LIN {X 0.098,Y -673.372,Z 1355.373,A 0.000,B 0.000,C 90.000,E1 103.175} C_DIS
LIN {X -0.021,Y -673.607,Z 1355.371,A 0.000,B 0.000,C 90.000,E1 102.703} C_DIS
LIN {X -0.341,Y -673.627,Z 1355.367,A 0.000,B 0.000,C 90.000,E1 102.007} C_DIS
LIN {X 0.141,Y -673.144,Z 1355.363,A 0.000,B 0.000,C 90.000,E1 101.243} C_DIS
LIN {X -0.111,Y -672.635,Z 1355.360,A 0.000,B 0.000,C 90.000,E1 100.782} C_DIS
LIN {X -0.239,Y -671.918,Z 1355.357,A 0.000,B 0.000,C 90.000,E1 100.310} C_DIS
LIN {X 0.170,Y -670.940,Z 1355.354,A 0.000,B 0.000,C 90.000,E1 99.792} C_DIS
LIN {X 0.024,Y -669.689,Z 1355.352,A 0.000,B 0.000,C 90.000,E1 99.321} C_DIS
LIN {X -0.238,Y -668.123,Z 1355.349,A 0.000,B 0.000,C 90.000,E1 98.859} C_DIS
LIN {X 0.063,Y -665.387,Z 1355.345,A 0.000,B 0.000,C 90.000,E1 98.106} C_DIS
LIN {X -0.221,Y -663.373,Z 1355.342,A 0.000,B 0.000,C 90.000,E1 97.644} C_DIS
LIN {X 0.125,Y -660.457,Z 1355.339,A 0.000,B 0.000,C 90.000,E1 97.004} C_DIS
LIN {X 0.159,Y -656.125,Z 1355.334,A 0.000,B 0.000,C 90.000,E1 96.144} C_DIS
LIN {X -0.289,Y -652.617,Z 1355.331,A 0.000,B 0.000,C 90.000,E1 95.568} C_DIS
LIN {X -0.279,Y -647.144,Z 1355.326,A 0.000,B 0.000,C 90.000,E1 94.702} C_DIS
LIN {X -0.203,Y -642.907,Z 1355.323,A 0.000,B 0.000,C 90.000,E1 94.073} C_DIS
LIN {X -0.112,Y -638.274,Z 1355.319,A 0.000,B 0.000,C 90.000,E1 93.440} C_DIS
LIN {X -0.068,Y -632.658,Z 1355.316,A 0.000,B 0.000,C 90.000,E1 92.808} C_DIS
LIN {X 0.041,Y -625.272,Z 1355.312,A 0.000,B 0.000,C 90.000,E1 92.064} C_DIS
LIN {X 0.162,Y -616.545,Z 1355.307,A 0.000,B 0.000,C 90.000,E1 91.203} C_DIS
LIN {X -0.082,Y -609.672,Z 1355.303,A 0.000,B 0.000,C 90.000,E1 90.630} C_DIS
LIN {X 0.197,Y -603.443,Z 1355.301,A 0.000,B 0.000,C 90.000,E1 90.172} C_DIS
LIN {X -0.078,Y -600.009,Z 1355.300,A 0.000,B 0.000,C 90.000,E1 90.000} C_DIS
LIN {X 0.088,Y -594.934,Z 1355.298,A 0.000,B 0.000,C 90.000,E1 89.714} C_DIS
LIN {X 0.288,Y -585.958,Z 1355.296,A 0.000,B 0.000,C 90.000,E1 89.312} C_DIS
LIN {X -0.105,Y -581.085,Z 1355.295,A 0.000,B 0.000,C 90.000,E1 89.141} C_DIS
LIN {X 0.058,Y -577.769,Z 1355.294,A 0.000,B 0.000,C 90.000,E1 88.969} C_DIS
LIN {X 0.028,Y -574.331,Z 1355.293,A 0.000,B 0.000,C 90.000,E1 88.740} C_DIS
LIN {X -0.031,Y -573.229,Z 1355.292,A 0.000,B 0.000,C 90.000,E1 88.568} C_DIS
LIN {X -0.073,Y -573.209,Z 1355.292,A 0.000,B 0.000,C 90.000,E1 88.568} C_DIS
LIN {X -0.166,Y -572.944,Z 1355.290,A 0.000,B 0.000,C 90.000,E1 88.224} C_DIS
LIN {X -0.181,Y -575.158,Z 1355.276,A 0.000,B 0.000,C 90.000,E1 85.641} C_DIS
LIN {X 0.153,Y -577.884,Z 1355.262,A 0.000,B 0.000,C 90.000,E1 83.166} C_DIS
LIN {X 0.133,Y -579.759,Z 1355.253,A 0.000,B 0.000,C 90.000,E1 81.546} C_DIS
LIN {X -0.211,Y -581.124,Z 1355.247,A 0.000,B 0.000,C 90.000,E1 80.500} C_DIS
LIN {X 0.269,Y -582.625,Z 1355.240,A 0.000,B 0.000,C 90.000,E1 79.106} C_DIS
LIN {X 0.312,Y -583.927,Z 1355.232,A 0.000,B 0.000,C 90.000,E1 77.757} C_DIS
LIN {X -0.190,Y -585.105,Z 1355.225,A 0.000,B 0.000,C 90.000,E1 76.464} C_DIS
LIN {X 0.210,Y -586.016,Z 1355.219,A 0.000,B 0.000,C 90.000,E1 75.353} C_DIS
LIN {X 0.198,Y -586.791,Z 1355.213,A 0.000,B 0.000,C 90.000,E1 74.283} C_DIS
LIN {X -0.190,Y -588.168,Z 1355.201,A 0.000,B 0.000,C 90.000,E1 72.181} C_DIS
LIN {X -0.025,Y -589.199,Z 1355.191,A 0.000,B 0.000,C 90.000,E1 70.296} C_DIS
LIN {X 0.180,Y -589.845,Z 1355.185,A 0.000,B 0.000,C 90.000,E1 69.209} C_DIS
LIN {X 0.038,Y -591.077,Z 1355.174,A 0.000,B 0.000,C 90.000,E1 67.358} C_DIS
LIN {X 0.054,Y -592.731,Z 1355.162,A 0.000,B 0.000,C 90.000,E1 65.229} C_DIS
LIN {X 0.108,Y -593.649,Z 1355.155,A 0.000,B 0.000,C 90.000,E1 63.896} C_DIS
LIN {X -0.357,Y -594.619,Z 1355.148,A 0.000,B 0.000,C 90.000,E1 62.615} C_DIS
LIN {X 0.103,Y -596.183,Z 1355.137,A 0.000,B 0.000,C 90.000,E1 60.717} C_DIS
LIN {X -0.005,Y -598.288,Z 1355.126,A 0.000,B 0.000,C 90.000,E1 58.614} C_DIS
LIN {X 0.140,Y -600.082,Z 1355.115,A 0.000,B 0.000,C 90.000,E1 56.755} C_DIS
LIN {X -0.059,Y -601.043,Z 1355.110,A 0.000,B 0.000,C 90.000,E1 55.722} C_DIS
LIN {X 0.000,Y -602.300,Z 1355.102,A 0.000,B 0.000,C 90.000,E1 54.402} C_DIS
LIN {X 0.068,Y -603.502,Z 1355.095,A 0.000,B 0.000,C 90.000,E1 53.084} C_DIS
LIN {X 0.140,Y -604.437,Z 1355.089,A 0.000,B 0.000,C 90.000,E1 52.029} C_DIS
LIN {X 0.125,Y -605.317,Z 1355.082,A 0.000,B 0.000,C 90.000,E1 50.723} C_DIS
LIN {X -0.351,Y -606.087,Z 1355.075,A 0.000,B 0.000,C 90.000,E1 49.461} C_DIS
LIN {X -0.228,Y -606.543,Z 1355.069,A 0.000,B 0.000,C 90.000,E1 48.405} C_DIS
LIN {X 0.114,Y -606.869,Z 1355.062,A 0.000,B 0.000,C 90.000,E1 47.067} C_DIS
LIN {X -0.393,Y -606.962,Z 1355.054,A 0.000,B 0.000,C 90.000,E1 45.810} C_DIS
LIN {X -0.288,Y -606.973,Z 1355.049,A 0.000,B 0.000,C 90.000,E1 44.757} C_DIS
LIN {X -0.186,Y -606.740,Z 1355.043,A 0.000,B 0.000,C 90.000,E1 43.704} C_DIS
LIN {X 0.157,Y -606.162,Z 1355.036,A 0.000,B 0.000,C 90.000,E1 42.366} C_DIS
LIN {X 0.081,Y -605.609,Z 1355.028,A 0.000,B 0.000,C 90.000,E1 41.067} C_DIS
LIN {X -0.081,Y -604.421,Z 1355.017,A 0.000,B 0.000,C 90.000,E1 38.991} C_DIS
LIN {X -0.101,Y -603.458,Z 1355.009,A 0.000,B 0.000,C 90.000,E1 37.684} C_DIS
LIN {X -0.140,Y -602.108,Z 1355.002,A 0.000,B 0.000,C 90.000,E1 36.377} C_DIS
LIN {X -0.224,Y -600.996,Z 1354.998,A 0.000,B 0.000,C 90.000,E1 35.598} C_DIS
LIN {X -0.079,Y -599.042,Z 1354.992,A 0.000,B 0.000,C 90.000,E1 34.532} C_DIS
LIN {X -0.303,Y -596.888,Z 1354.986,A 0.000,B 0.000,C 90.000,E1 33.499} C_DIS
LIN {X 0.160,Y -593.675,Z 1354.979,A 0.000,B 0.000,C 90.000,E1 32.133} C_DIS
LIN {X 0.264,Y -592.209,Z 1354.976,A 0.000,B 0.000,C 90.000,E1 31.592} C_DIS
LIN {X 0.137,Y -588.654,Z 1354.970,A 0.000,B 0.000,C 90.000,E1 30.541} C_DIS
LIN {X 0.089,Y -585.811,Z 1354.965,A 0.000,B 0.000,C 90.000,E1 29.745} C_DIS
LIN {X 0.136,Y -583.669,Z 1354.962,A 0.000,B 0.000,C 90.000,E1 29.205} C_DIS
LIN {X -0.109,Y -578.764,Z 1354.956,A 0.000,B 0.000,C 90.000,E1 28.153} C_DIS
LIN {X 0.078,Y -573.243,Z 1354.950,A 0.000,B 0.000,C 90.000,E1 27.052} C_DIS
LIN {X 0.182,Y -569.449,Z 1354.947,A 0.000,B 0.000,C 90.000,E1 26.360} C_DIS
LIN {X -0.250,Y -565.264,Z 1354.943,A 0.000,B 0.000,C 90.000,E1 25.720} C_DIS
LIN {X -0.111,Y -561.716,Z 1354.940,A 0.000,B 0.000,C 90.000,E1 25.155} C_DIS
LIN {X 0.004,Y -557.868,Z 1354.937,A 0.000,B 0.000,C 90.000,E1 24.591} C_DIS
LIN {X -0.129,Y -551.792,Z 1354.932,A 0.000,B 0.000,C 90.000,E1 23.770} C_DIS
LIN {X -0.206,Y -546.341,Z 1354.928,A 0.000,B 0.000,C 90.000,E1 23.078} C_DIS
LIN {X -0.074,Y -542.890,Z 1354.926,A 0.000,B 0.000,C 90.000,E1 22.642} C_DIS
LIN {X 0.139,Y -532.965,Z 1354.919,A 0.000,B 0.000,C 90.000,E1 21.482} C_DIS
LIN {X -0.080,Y -524.058,Z 1354.914,A 0.000,B 0.000,C 90.000,E1 20.536} C_DIS
LIN {X 0.210,Y -512.237,Z 1354.907,A 0.000,B 0.000,C 90.000,E1 19.268} C_DIS
LIN {X 0.003,Y -502.949,Z 1354.902,A 0.000,B 0.000,C 90.000,E1 18.308} C_DIS
LIN {X 0.037,Y -493.704,Z 1354.896,A 0.000,B 0.000,C 90.000,E1 17.347} C_DIS
LIN {X 0.061,Y -483.571,Z 1354.891,A 0.000,B 0.000,C 90.000,E1 16.386} C_DIS
LIN {X -0.235,Y -470.744,Z 1354.884,A 0.000,B 0.000,C 90.000,E1 15.190} C_DIS
LIN {X -0.084,Y -459.483,Z 1354.878,A 0.000,B 0.000,C 90.000,E1 14.064} C_DIS
LIN {X -0.197,Y -439.447,Z 1354.867,A 0.000,B 0.000,C 90.000,E1 12.063} C_DIS
LIN {X 0.044,Y -422.530,Z 1354.857,A 0.000,B 0.000,C 90.000,E1 10.197} C_DIS
LIN {X -0.139,Y -408.504,Z 1354.848,A 0.000,B 0.000,C 90.000,E1 8.624} C_DIS
LIN {X -0.093,Y -399.960,Z 1354.842,A 0.000,B 0.000,C 90.000,E1 7.644} C_DIS
LIN {X -0.002,Y -397.197,Z 1354.841,A 0.000,B 0.000,C 90.000,E1 7.296} C_DIS
LIN {X 0.091,Y -393.893,Z 1354.838,A 0.000,B 0.000,C 90.000,E1 6.777} C_DIS
LIN {X 0.053,Y -393.861,Z 1354.838,A 0.000,B 0.000,C 90.000,E1 6.777} C_DIS
LIN {X -0.024,Y -394.940,Z 1354.837,A 0.000,B 0.000,C 90.000,E1 6.606} C_DIS
LIN {X -0.066,Y -398.783,Z 1354.835,A 0.000,B 0.000,C 90.000,E1 6.258} C_DIS
LIN {X 0.058,Y -412.298,Z 1354.829,A 0.000,B 0.000,C 90.000,E1 5.277} C_DIS
LIN {X -0.119,Y -417.007,Z 1354.827,A 0.000,B 0.000,C 90.000,E1 4.935} C_DIS
LIN {X 0.172,Y -423.162,Z 1354.824,A 0.000,B 0.000,C 90.000,E1 4.359} C_DIS
LIN {X 0.210,Y -428.896,Z 1354.821,A 0.000,B 0.000,C 90.000,E1 3.784} C_DIS
LIN {X -0.032,Y -434.486,Z 1354.818,A 0.000,B 0.000,C 90.000,E1 3.212} C_DIS
LIN {X 0.147,Y -441.264,Z 1354.813,A 0.000,B 0.000,C 90.000,E1 2.407} C_DIS
LIN {X 0.130,Y -447.486,Z 1354.809,A 0.000,B 0.000,C 90.000,E1 1.661} C_DIS
LIN {X 0.087,Y -453.726,Z 1354.805,A 0.000,B 0.000,C 90.000,E1 0.859} C_DIS
LIN {X -0.019,Y -458.436,Z 1354.801,A 0.000,B 0.000,C 90.000,E1 0.229} C_DIS
LIN {X 0.021,Y -464.684,Z 1354.796,A 0.000,B 0.000,C 90.000,E1 359.312} C_DIS
LIN {X 0.111,Y -469.753,Z 1354.792,A 0.000,B 0.000,C 90.000,E1 358.511} C_DIS
LIN {X -0.204,Y -474.343,Z 1354.787,A 0.000,B 0.000,C 90.000,E1 357.764} C_DIS
LIN {X -0.025,Y -478.713,Z 1354.783,A 0.000,B 0.000,C 90.000,E1 356.963} C_DIS
LIN {X 0.223,Y -482.743,Z 1354.779,A 0.000,B 0.000,C 90.000,E1 356.159} C_DIS
LIN {X -0.121,Y -485.731,Z 1354.775,A 0.000,B 0.000,C 90.000,E1 355.584} C_DIS
LIN {X -0.133,Y -489.757,Z 1354.770,A 0.000,B 0.000,C 90.000,E1 354.666} C_DIS
LIN {X -0.102,Y -491.688,Z 1354.768,A 0.000,B 0.000,C 90.000,E1 354.204} C_DIS
LIN {X -0.003,Y -495.070,Z 1354.763,A 0.000,B 0.000,C 90.000,E1 353.280} C_DIS
LIN {X 0.135,Y -498.250,Z 1354.758,A 0.000,B 0.000,C 90.000,E1 352.356} C_DIS
LIN {X 0.047,Y -499.271,Z 1354.756,A 0.000,B 0.000,C 90.000,E1 352.064} C_DIS
LIN {X 0.232,Y -501.799,Z 1354.751,A 0.000,B 0.000,C 90.000,E1 351.141} C_DIS
LIN {X -0.120,Y -504.896,Z 1354.744,A 0.000,B 0.000,C 90.000,E1 349.982} C_DIS
LIN {X 0.155,Y -507.585,Z 1354.738,A 0.000,B 0.000,C 90.000,E1 348.757} C_DIS
LIN {X 0.014,Y -509.380,Z 1354.733,A 0.000,B 0.000,C 90.000,E1 347.881} C_DIS
LIN {X 0.004,Y -510.932,Z 1354.728,A 0.000,B 0.000,C 90.000,E1 346.992} C_DIS
LIN {X -0.013,Y -512.701,Z 1354.721,A 0.000,B 0.000,C 90.000,E1 345.811} C_DIS
LIN {X -0.109,Y -513.853,Z 1354.716,A 0.000,B 0.000,C 90.000,E1 344.936} C_DIS
LIN {X 0.074,Y -514.747,Z 1354.711,A 0.000,B 0.000,C 90.000,E1 344.031} C_DIS
LIN {X 0.130,Y -515.354,Z 1354.706,A 0.000,B 0.000,C 90.000,E1 343.142} C_DIS
LIN {X -0.185,Y -515.684,Z 1354.700,A 0.000,B 0.000,C 90.000,E1 342.000} C_DIS
LIN {X -0.060,Y -515.743,Z 1354.698,A 0.000,B 0.000,C 90.000,E1 341.692} C_DIS
LIN {X -0.096,Y -515.674,Z 1354.697,A 0.000,B 0.000,C 90.000,E1 341.402} C_DIS
LIN {X 0.030,Y -515.467,Z 1354.695,A 0.000,B 0.000,C 90.000,E1 341.094} C_DIS
LIN {X 0.159,Y -515.103,Z 1354.693,A 0.000,B 0.000,C 90.000,E1 340.786} C_DIS
LIN {X 0.114,Y -514.518,Z 1354.692,A 0.000,B 0.000,C 90.000,E1 340.496} C_DIS
LIN {X -0.244,Y -513.577,Z 1354.690,A 0.000,B 0.000,C 90.000,E1 340.242} C_DIS
LIN {X 0.060,Y -512.867,Z 1354.689,A 0.000,B 0.000,C 90.000,E1 340.061} C_DIS
LIN {X -0.119,Y -511.804,Z 1354.688,A 0.000,B 0.000,C 90.000,E1 339.934} C_DIS
LIN {X 0.181,Y -509.106,Z 1354.688,A 0.000,B 0.000,C 90.000,E1 339.752} C_DIS
LIN {X 0.170,Y -478.324,Z 1354.680,A 0.000,B 0.000,C 90.000,E1 338.411} C_DIS
LIN {X 0.089,Y -449.677,Z 1354.672,A 0.000,B 0.000,C 90.000,E1 336.997} C_DIS
LIN {X -0.133,Y -424.639,Z 1354.664,A 0.000,B 0.000,C 90.000,E1 335.613} C_DIS
LIN {X -0.216,Y -401.544,Z 1354.656,A 0.000,B 0.000,C 90.000,E1 334.152} C_DIS
LIN {X -0.114,Y -380.373,Z 1354.648,A 0.000,B 0.000,C 90.000,E1 332.615} C_DIS
LIN {X 0.040,Y -366.210,Z 1354.642,A 0.000,B 0.000,C 90.000,E1 331.463} C_DIS
LIN {X 0.013,Y -366.169,Z 1354.641,A 0.000,B 0.000,C 90.000,E1 331.463} C_DIS
LIN {X 0.084,Y -371.188,Z 1354.604,A 0.000,B 0.000,C 90.000,E1 324.769} C_DIS
LIN {X 0.071,Y -371.620,Z 1354.602,A 0.000,B 0.000,C 90.000,E1 324.402} C_DIS
LIN {X -0.121,Y -376.725,Z 1354.570,A 0.000,B 0.000,C 90.000,E1 318.566} C_DIS
LIN {X -0.117,Y -378.122,Z 1354.564,A 0.000,B 0.000,C 90.000,E1 317.472} C_DIS
LIN {X -0.096,Y -384.239,Z 1354.529,A 0.000,B 0.000,C 90.000,E1 311.310} C_DIS
LIN {X -0.052,Y -384.743,Z 1354.527,A 0.000,B 0.000,C 90.000,E1 310.943} C_DIS
LIN {X 0.191,Y -390.909,Z 1354.494,A 0.000,B 0.000,C 90.000,E1 304.818} C_DIS
LIN {X 0.037,Y -391.347,Z 1354.492,A 0.000,B 0.000,C 90.000,E1 304.485} C_DIS
LIN {X -0.140,Y -397.058,Z 1354.458,A 0.000,B 0.000,C 90.000,E1 298.487} C_DIS
LIN {X 0.165,Y -401.450,Z 1354.427,A 0.000,B 0.000,C 90.000,E1 292.823} C_DIS
LIN {X -0.125,Y -401.677,Z 1354.425,A 0.000,B 0.000,C 90.000,E1 292.514} C_DIS
LIN {X -0.095,Y -404.537,Z 1354.396,A 0.000,B 0.000,C 90.000,E1 287.275} C_DIS
LIN {X 0.005,Y -404.763,Z 1354.394,A 0.000,B 0.000,C 90.000,E1 286.913} C_DIS
LIN {X -0.088,Y -406.150,Z 1354.363,A 0.000,B 0.000,C 90.000,E1 281.366} C_DIS
LIN {X 0.016,Y -405.648,Z 1354.334,A 0.000,B 0.000,C 90.000,E1 276.144} C_DIS
LIN {X 0.021,Y -405.625,Z 1354.332,A 0.000,B 0.000,C 90.000,E1 275.796} C_DIS
LIN {X 0.094,Y -403.554,Z 1354.305,A 0.000,B 0.000,C 90.000,E1 270.917} C_DIS
LIN {X 0.029,Y -403.075,Z 1354.301,A 0.000,B 0.000,C 90.000,E1 270.229} C_DIS
LIN {X -0.144,Y -399.024,Z 1354.272,A 0.000,B 0.000,C 90.000,E1 265.008} C_DIS
LIN {X 0.169,Y -398.149,Z 1354.268,A 0.000,B 0.000,C 90.000,E1 264.261} C_DIS
LIN {X 0.027,Y -392.946,Z 1354.241,A 0.000,B 0.000,C 90.000,E1 259.342} C_DIS
LIN {X -0.015,Y -392.509,Z 1354.239,A 0.000,B 0.000,C 90.000,E1 258.993} C_DIS
LIN {X 0.132,Y -386.143,Z 1354.213,A 0.000,B 0.000,C 90.000,E1 254.338} C_DIS
LIN {X 0.092,Y -385.021,Z 1354.207,A 0.000,B 0.000,C 90.000,E1 253.268} C_DIS
LIN {X -0.036,Y -378.156,Z 1354.183,A 0.000,B 0.000,C 90.000,E1 248.954} C_DIS
LIN {X 0.179,Y -375.917,Z 1354.173,A 0.000,B 0.000,C 90.000,E1 247.102} C_DIS
LIN {X -0.201,Y -369.131,Z 1354.151,A 0.000,B 0.000,C 90.000,E1 243.127} C_DIS
LIN {X 0.028,Y -366.281,Z 1354.138,A 0.000,B 0.000,C 90.000,E1 240.873} C_DIS
LIN {X 0.103,Y -358.367,Z 1354.111,A 0.000,B 0.000,C 90.000,E1 236.008} C_DIS
LIN {X 0.154,Y -356.064,Z 1354.101,A 0.000,B 0.000,C 90.000,E1 234.116} C_DIS
LIN {X -0.114,Y -348.502,Z 1354.073,A 0.000,B 0.000,C 90.000,E1 229.218} C_DIS
LIN {X -0.042,Y -345.927,Z 1354.061,A 0.000,B 0.000,C 90.000,E1 226.905} C_DIS
LIN {X 0.176,Y -339.143,Z 1354.033,A 0.000,B 0.000,C 90.000,E1 221.838} C_DIS
LIN {X 0.045,Y -336.972,Z 1354.020,A 0.000,B 0.000,C 90.000,E1 219.519} C_DIS
LIN {X -0.056,Y -334.991,Z 1354.011,A 0.000,B 0.000,C 90.000,E1 217.971} C_DIS
LIN {X 0.146,Y -329.803,Z 1353.980,A 0.000,B 0.000,C 90.000,E1 212.339} C_DIS
LIN {X 0.128,Y -329.802,Z 1353.980,A 0.000,B 0.000,C 90.000,E1 212.339} C_DIS
LIN {X 0.133,Y -347.212,Z 1353.970,A 0.000,B 0.000,C 90.000,E1 210.590} C_DIS
LIN {X 0.036,Y -366.706,Z 1353.960,A 0.000,B 0.000,C 90.000,E1 208.871} C_DIS
LIN {X -0.108,Y -388.168,Z 1353.951,A 0.000,B 0.000,C 90.000,E1 207.206} C_DIS
LIN {X 0.075,Y -409.913,Z 1353.943,A 0.000,B 0.000,C 90.000,E1 205.668} C_DIS
LIN {X 0.080,Y -433.617,Z 1353.935,A 0.000,B 0.000,C 90.000,E1 204.207} C_DIS
LIN {X 0.228,Y -445.571,Z 1353.931,A 0.000,B 0.000,C 90.000,E1 203.515} C_DIS
LIN {X 0.188,Y -448.362,Z 1353.930,A 0.000,B 0.000,C 90.000,E1 203.334} C_DIS
LIN {X 0.072,Y -449.801,Z 1353.929,A 0.000,B 0.000,C 90.000,E1 203.131} C_DIS
LIN {X -0.054,Y -451.172,Z 1353.927,A 0.000,B 0.000,C 90.000,E1 202.823} C_DIS
LIN {X -0.172,Y -452.149,Z 1353.925,A 0.000,B 0.000,C 90.000,E1 202.514} C_DIS
LIN {X 0.132,Y -452.930,Z 1353.923,A 0.000,B 0.000,C 90.000,E1 202.153} C_DIS
LIN {X 0.022,Y -453.562,Z 1353.921,A 0.000,B 0.000,C 90.000,E1 201.844} C_DIS
LIN {X -0.190,Y -454.472,Z 1353.918,A 0.000,B 0.000,C 90.000,E1 201.227} C_DIS
LIN {X -0.171,Y -455.790,Z 1353.911,A 0.000,B 0.000,C 90.000,E1 199.939} C_DIS
LIN {X -0.143,Y -458.039,Z 1353.898,A 0.000,B 0.000,C 90.000,E1 197.692} C_DIS
LIN {X -0.020,Y -459.483,Z 1353.889,A 0.000,B 0.000,C 90.000,E1 196.079} C_DIS
LIN {X -0.090,Y -461.017,Z 1353.879,A 0.000,B 0.000,C 90.000,E1 194.175} C_DIS
LIN {X -0.141,Y -462.346,Z 1353.870,A 0.000,B 0.000,C 90.000,E1 192.591} C_DIS
LIN {X -0.115,Y -464.243,Z 1353.858,A 0.000,B 0.000,C 90.000,E1 190.366} C_DIS
LIN {X 0.186,Y -465.365,Z 1353.849,A 0.000,B 0.000,C 90.000,E1 188.746} C_DIS
LIN {X 0.052,Y -465.966,Z 1353.844,A 0.000,B 0.000,C 90.000,E1 187.814} C_DIS
LIN {X 0.067,Y -466.673,Z 1353.836,A 0.000,B 0.000,C 90.000,E1 186.549} C_DIS
LIN {X -0.100,Y -467.163,Z 1353.828,A 0.000,B 0.000,C 90.000,E1 184.992} C_DIS
LIN {X 0.177,Y -467.337,Z 1353.823,A 0.000,B 0.000,C 90.000,E1 184.012} C_DIS
LIN {X -0.048,Y -467.393,Z 1353.817,A 0.000,B 0.000,C 90.000,E1 183.094} C_DIS
LIN {X 0.175,Y -467.312,Z 1353.812,A 0.000,B 0.000,C 90.000,E1 182.121} C_DIS
LIN {X -0.050,Y -467.109,Z 1353.807,A 0.000,B 0.000,C 90.000,E1 181.203} C_DIS
LIN {X 0.176,Y -466.538,Z 1353.801,A 0.000,B 0.000,C 90.000,E1 180.229} C_DIS
LIN {X 0.169,Y -466.028,Z 1353.798,A 0.000,B 0.000,C 90.000,E1 179.599} C_DIS
LIN {X -0.084,Y -464.912,Z 1353.793,A 0.000,B 0.000,C 90.000,E1 178.682} C_DIS
LIN {X 0.128,Y -463.685,Z 1353.787,A 0.000,B 0.000,C 90.000,E1 177.707} C_DIS
LIN {X 0.095,Y -462.675,Z 1353.784,A 0.000,B 0.000,C 90.000,E1 177.078} C_DIS
LIN {X -0.179,Y -460.650,Z 1353.779,A 0.000,B 0.000,C 90.000,E1 176.159} C_DIS
LIN {X -0.209,Y -459.147,Z 1353.775,A 0.000,B 0.000,C 90.000,E1 175.527} C_DIS
LIN {X 0.208,Y -457.534,Z 1353.771,A 0.000,B 0.000,C 90.000,E1 174.837} C_DIS
LIN {X -0.214,Y -454.731,Z 1353.767,A 0.000,B 0.000,C 90.000,E1 174.090} C_DIS
LIN {X -0.162,Y -451.422,Z 1353.763,A 0.000,B 0.000,C 90.000,E1 173.280} C_DIS
LIN {X 0.179,Y -448.396,Z 1353.759,A 0.000,B 0.000,C 90.000,E1 172.591} C_DIS
LIN {X -0.013,Y -445.899,Z 1353.756,A 0.000,B 0.000,C 90.000,E1 172.129} C_DIS
LIN {X -0.049,Y -441.166,Z 1353.752,A 0.000,B 0.000,C 90.000,E1 171.319} C_DIS
LIN {X -0.027,Y -434.660,Z 1353.746,A 0.000,B 0.000,C 90.000,E1 170.330} C_DIS
LIN {X -0.079,Y -427.731,Z 1353.741,A 0.000,B 0.000,C 90.000,E1 169.342} C_DIS
LIN {X 0.199,Y -411.920,Z 1353.728,A 0.000,B 0.000,C 90.000,E1 166.937} C_DIS
LIN {X 0.022,Y -404.485,Z 1353.721,A 0.000,B 0.000,C 90.000,E1 165.755} C_DIS
LIN {X 0.069,Y -401.861,Z 1353.718,A 0.000,B 0.000,C 90.000,E1 165.227} C_DIS
LIN {X 0.237,Y -400.509,Z 1353.716,A 0.000,B 0.000,C 90.000,E1 164.866} C_DIS
LIN {X -0.143,Y -400.022,Z 1353.715,A 0.000,B 0.000,C 90.000,E1 164.755} C_DIS
LIN {X -0.031,Y -399.728,Z 1353.714,A 0.000,B 0.000,C 90.000,E1 164.574} C_DIS
LIN {X 0.048,Y -399.581,Z 1353.711,A 0.000,B 0.000,C 90.000,E1 164.031} C_DIS
LIN {X 0.009,Y -399.582,Z 1353.711,A 0.000,B 0.000,C 90.000,E1 164.031} C_DIS
LIN {X 0.016,Y -400.248,Z 1353.710,A 0.000,B 0.000,C 90.000,E1 163.866} C_DIS
LIN {X -0.084,Y -405.513,Z 1353.707,A 0.000,B 0.000,C 90.000,E1 163.196} C_DIS
LIN {X 0.081,Y -411.201,Z 1353.703,A 0.000,B 0.000,C 90.000,E1 162.598} C_DIS
LIN {X 0.103,Y -419.234,Z 1353.699,A 0.000,B 0.000,C 90.000,E1 161.873} C_DIS
LIN {X -0.100,Y -439.980,Z 1353.690,A 0.000,B 0.000,C 90.000,E1 160.242} C_DIS
LIN {X 0.004,Y -455.872,Z 1353.684,A 0.000,B 0.000,C 90.000,E1 159.028} C_DIS
END
